// TIA Portal V17 export
// export: Created 2025-03-07T09:19:05.4245713Z, ExportSetting WithDefaults, DisplayName Totally Integrated Automation Portal, DisplayVersion V17 Update 8, DisplayName TIA Portal Openness, DisplayVersion V17 Update 8, DisplayName TIA Portal Version Control Interface, DisplayVersion V17, DisplayName SINAMICS Startdrive Advanced, DisplayVersion V17 SP2, DisplayName SINAMICS Startdrive G110M, G120, G120C, G120D, G120P, G115D, DisplayVersion V17 SP2, DisplayName SINAMICS Startdrive G130, G150, S120, S150, SINAMICS MV, S210, DisplayVersion V17 SP2, DisplayName STEP 7 Professional, DisplayVersion V17 Update 8, DisplayName SINUMERIK ONE STEP 7 Toolbox, DisplayVersion V17 Update 12, DisplayName SINUMERIK 840D sl STEP 7 Toolbox, DisplayVersion V17 Update 12, DisplayName STEP 7 Safety, DisplayVersion V17 Update 6, DisplayName WinCC Advanced, DisplayVersion V17 Update 8
FUNCTION "FC16701_OPC_UA_MASTER_MACHINE_DATA_UPDATE" : Void   // FC16701, LAD
{ S7_Optimized_Access := 'TRUE' }
VERSION : 0.1
// stored: AutoNumber false, IsIECCheckEnabled false, SetENOAutomatically false, UDAEnableTagReadback false
   VAR_TEMP
      RETVAL : Word;
      U01_ASPIRATION_FINAL_VALUE_AUX : Real;
      U02_ASPIRATION_FINAL_VALUE_AUX : Real;
   END_VAR
   VAR_TEMP   // added for the SCL form of the ladder/FBD networks
      _w1 : Bool;
      _w2 : Bool;
      _w3 : Bool;
      _w4 : Bool;
      _w5 : Bool;
   END_VAR
BEGIN

REGION Network 1: <<<<<<<<<<<<<<<<<<<< OPC UA MASTER MACHINE >>>>>>>>>>>>>>>>>>>>
END_REGION

REGION Network 2: GENERAL INFO - ID
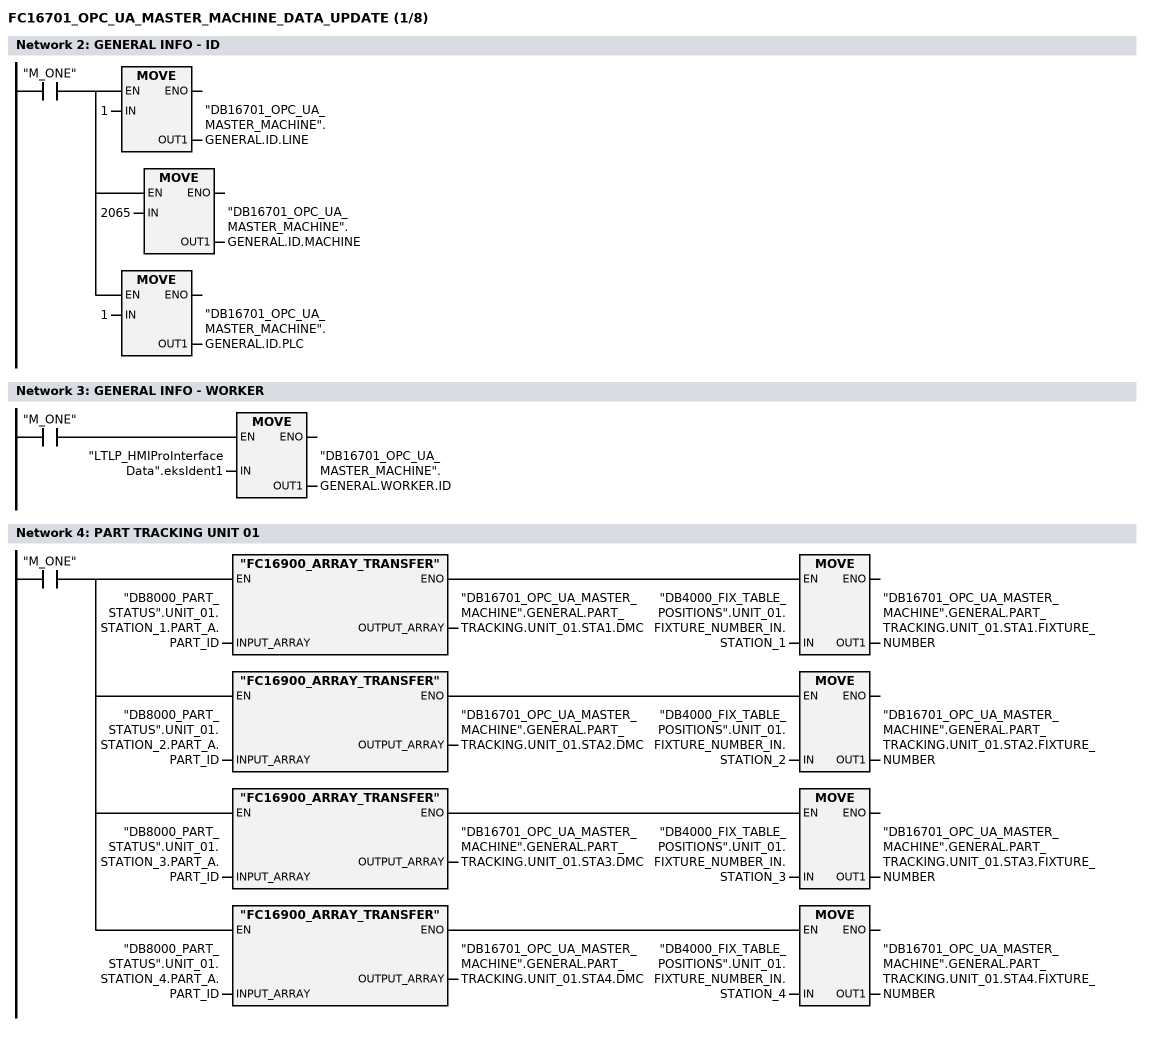
   RUNG wire#powerrail
      Contact( "M_ONE" )
      wire#w1
      Move(in := 1, out1 => "DB16701_OPC_UA_MASTER_MACHINE".GENERAL.ID.LINE)
   END_RUNG
   RUNG wire#w1
      Move(in := 2065, out1 => "DB16701_OPC_UA_MASTER_MACHINE".GENERAL.ID.MACHINE)
   END_RUNG
   RUNG wire#w1
      Move(in := 1, out1 => "DB16701_OPC_UA_MASTER_MACHINE".GENERAL.ID.PLC)
   END_RUNG
   // the same network as SCL:
   IF "M_ONE" THEN
       "DB16701_OPC_UA_MASTER_MACHINE".GENERAL.ID.LINE := 1;
       "DB16701_OPC_UA_MASTER_MACHINE".GENERAL.ID.MACHINE := 2065;
       "DB16701_OPC_UA_MASTER_MACHINE".GENERAL.ID.PLC := 1;
   END_IF;
END_REGION

REGION Network 3: GENERAL INFO - WORKER
   RUNG wire#powerrail
      Contact( "M_ONE" )
      Move(in := "LTLP_HMIProInterfaceData".eksIdent1, out1 => "DB16701_OPC_UA_MASTER_MACHINE".GENERAL.WORKER.ID)
   END_RUNG
   // the same network as SCL:
   IF "M_ONE" THEN
       "DB16701_OPC_UA_MASTER_MACHINE".GENERAL.WORKER.ID := "LTLP_HMIProInterfaceData".eksIdent1;
   END_IF;
END_REGION

REGION Network 4: PART TRACKING UNIT 01
   RUNG wire#powerrail
      Contact( "M_ONE" )
      wire#w1
      "FC16900_ARRAY_TRANSFER"(INPUT_ARRAY := "DB8000_PART_STATUS".UNIT_01.STATION_1.PART_A.PART_ID, OUTPUT_ARRAY => "DB16701_OPC_UA_MASTER_MACHINE".GENERAL.PART_TRACKING.UNIT_01.STA1.DMC)
      Move(in := "DB4000_FIX_TABLE_POSITIONS".UNIT_01.FIXTURE_NUMBER_IN.STATION_1, out1 => "DB16701_OPC_UA_MASTER_MACHINE".GENERAL.PART_TRACKING.UNIT_01.STA1.FIXTURE_NUMBER)
   END_RUNG
   RUNG wire#w1
      "FC16900_ARRAY_TRANSFER"(INPUT_ARRAY := "DB8000_PART_STATUS".UNIT_01.STATION_2.PART_A.PART_ID, OUTPUT_ARRAY => "DB16701_OPC_UA_MASTER_MACHINE".GENERAL.PART_TRACKING.UNIT_01.STA2.DMC)
      Move(in := "DB4000_FIX_TABLE_POSITIONS".UNIT_01.FIXTURE_NUMBER_IN.STATION_2, out1 => "DB16701_OPC_UA_MASTER_MACHINE".GENERAL.PART_TRACKING.UNIT_01.STA2.FIXTURE_NUMBER)
   END_RUNG
   RUNG wire#w1
      "FC16900_ARRAY_TRANSFER"(INPUT_ARRAY := "DB8000_PART_STATUS".UNIT_01.STATION_3.PART_A.PART_ID, OUTPUT_ARRAY => "DB16701_OPC_UA_MASTER_MACHINE".GENERAL.PART_TRACKING.UNIT_01.STA3.DMC)
      Move(in := "DB4000_FIX_TABLE_POSITIONS".UNIT_01.FIXTURE_NUMBER_IN.STATION_3, out1 => "DB16701_OPC_UA_MASTER_MACHINE".GENERAL.PART_TRACKING.UNIT_01.STA3.FIXTURE_NUMBER)
   END_RUNG
   RUNG wire#w1
      "FC16900_ARRAY_TRANSFER"(INPUT_ARRAY := "DB8000_PART_STATUS".UNIT_01.STATION_4.PART_A.PART_ID, OUTPUT_ARRAY => "DB16701_OPC_UA_MASTER_MACHINE".GENERAL.PART_TRACKING.UNIT_01.STA4.DMC)
      Move(in := "DB4000_FIX_TABLE_POSITIONS".UNIT_01.FIXTURE_NUMBER_IN.STATION_4, out1 => "DB16701_OPC_UA_MASTER_MACHINE".GENERAL.PART_TRACKING.UNIT_01.STA4.FIXTURE_NUMBER)
   END_RUNG
   // the same network as SCL:
   #_w2 := "M_ONE";
   "FC16900_ARRAY_TRANSFER"(EN := "M_ONE",
                           INPUT_ARRAY := "DB8000_PART_STATUS".UNIT_01.STATION_1.PART_A.PART_ID,
                           OUTPUT_ARRAY => "DB16701_OPC_UA_MASTER_MACHINE".GENERAL.PART_TRACKING.UNIT_01.STA1.DMC,
                           ENO => #_w1);
   IF #_w1 THEN
       "DB16701_OPC_UA_MASTER_MACHINE".GENERAL.PART_TRACKING.UNIT_01.STA1.FIXTURE_NUMBER := "DB4000_FIX_TABLE_POSITIONS".UNIT_01.FIXTURE_NUMBER_IN.STATION_1;
   END_IF;
   "FC16900_ARRAY_TRANSFER"(EN := #_w2,
                           INPUT_ARRAY := "DB8000_PART_STATUS".UNIT_01.STATION_2.PART_A.PART_ID,
                           OUTPUT_ARRAY => "DB16701_OPC_UA_MASTER_MACHINE".GENERAL.PART_TRACKING.UNIT_01.STA2.DMC,
                           ENO => #_w3);
   IF #_w3 THEN
       "DB16701_OPC_UA_MASTER_MACHINE".GENERAL.PART_TRACKING.UNIT_01.STA2.FIXTURE_NUMBER := "DB4000_FIX_TABLE_POSITIONS".UNIT_01.FIXTURE_NUMBER_IN.STATION_2;
   END_IF;
   "FC16900_ARRAY_TRANSFER"(EN := #_w2,
                           INPUT_ARRAY := "DB8000_PART_STATUS".UNIT_01.STATION_3.PART_A.PART_ID,
                           OUTPUT_ARRAY => "DB16701_OPC_UA_MASTER_MACHINE".GENERAL.PART_TRACKING.UNIT_01.STA3.DMC,
                           ENO => #_w4);
   IF #_w4 THEN
       "DB16701_OPC_UA_MASTER_MACHINE".GENERAL.PART_TRACKING.UNIT_01.STA3.FIXTURE_NUMBER := "DB4000_FIX_TABLE_POSITIONS".UNIT_01.FIXTURE_NUMBER_IN.STATION_3;
   END_IF;
   "FC16900_ARRAY_TRANSFER"(EN := #_w2,
                           INPUT_ARRAY := "DB8000_PART_STATUS".UNIT_01.STATION_4.PART_A.PART_ID,
                           OUTPUT_ARRAY => "DB16701_OPC_UA_MASTER_MACHINE".GENERAL.PART_TRACKING.UNIT_01.STA4.DMC,
                           ENO => #_w5);
   IF #_w5 THEN
       "DB16701_OPC_UA_MASTER_MACHINE".GENERAL.PART_TRACKING.UNIT_01.STA4.FIXTURE_NUMBER := "DB4000_FIX_TABLE_POSITIONS".UNIT_01.FIXTURE_NUMBER_IN.STATION_4;
   END_IF;
END_REGION

REGION Network 5: PART TRACKING UNIT 02
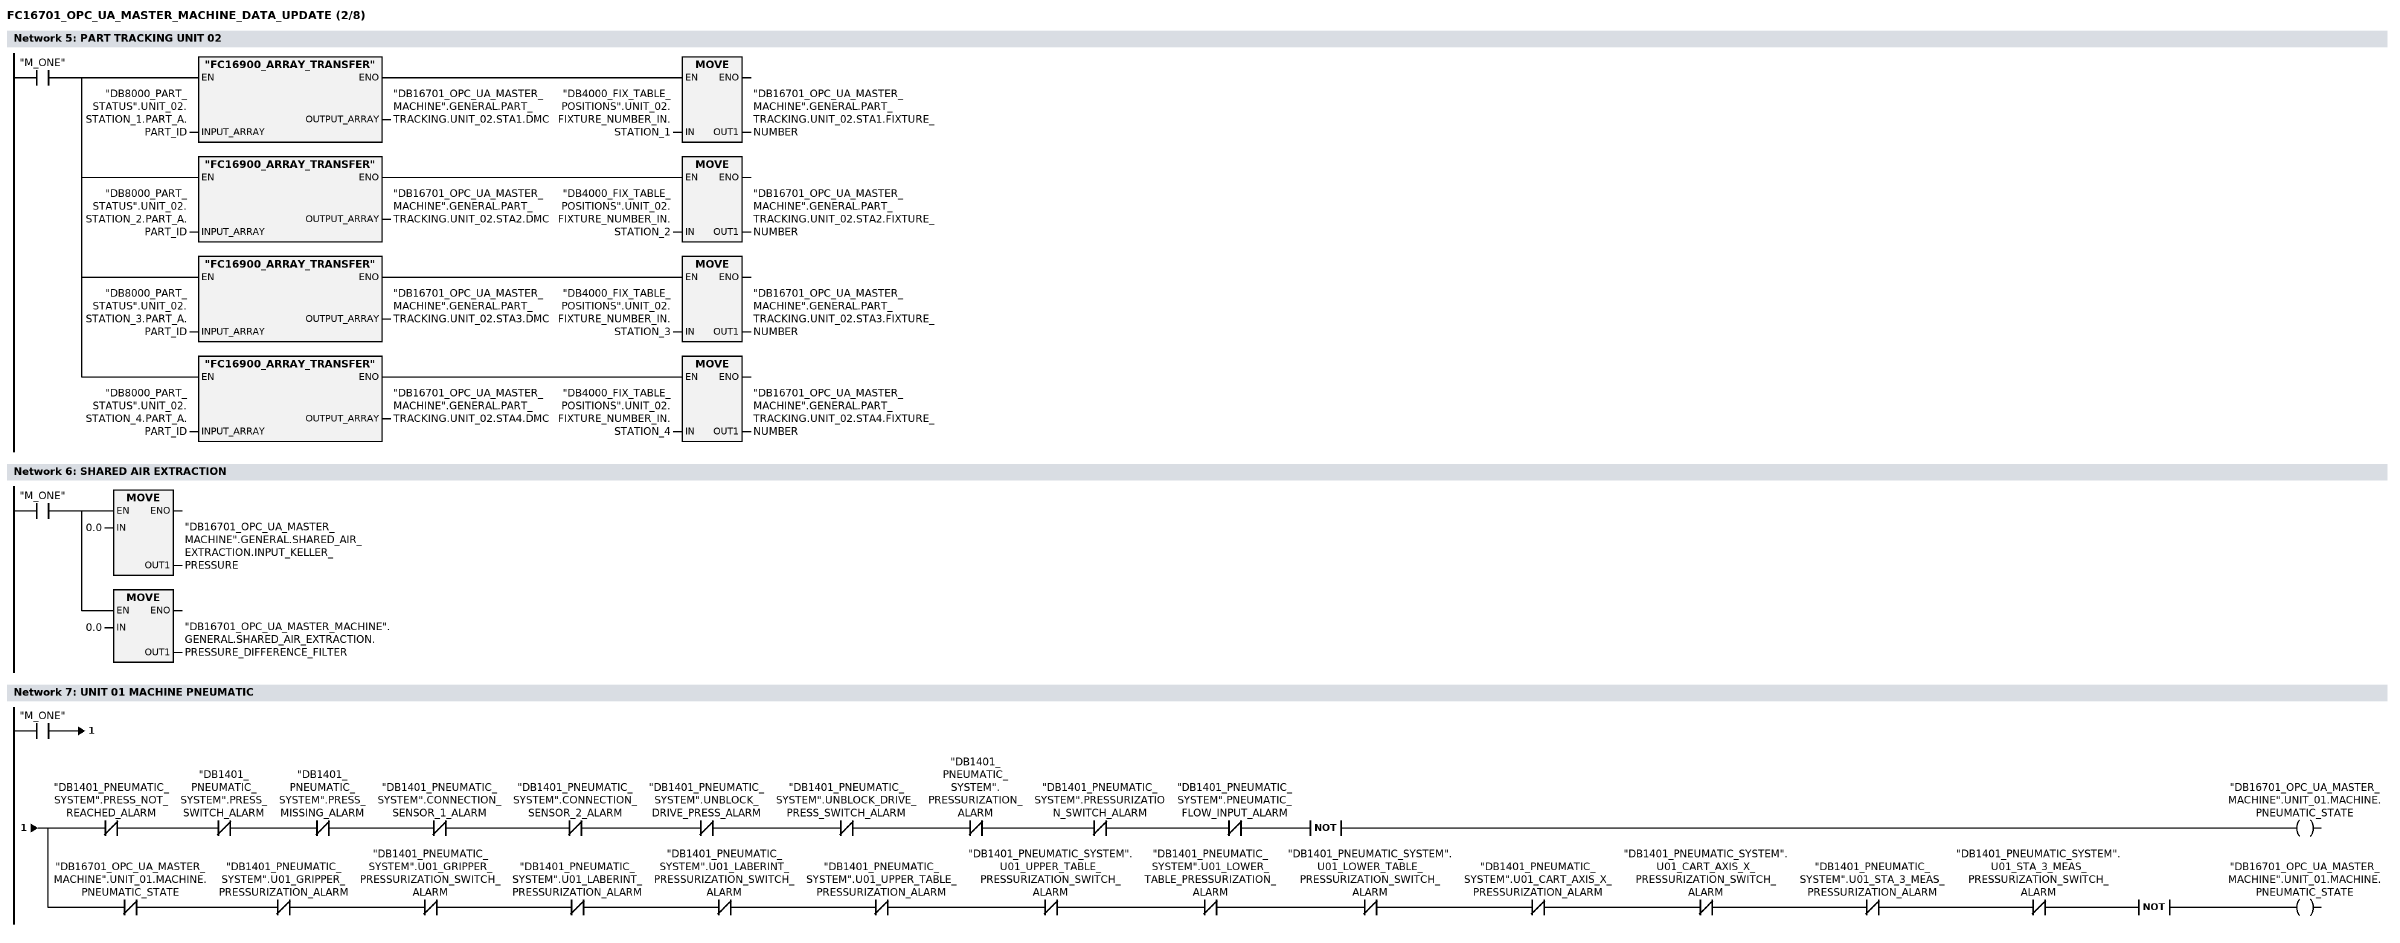
   RUNG wire#powerrail
      Contact( "M_ONE" )
      wire#w1
      "FC16900_ARRAY_TRANSFER"(INPUT_ARRAY := "DB8000_PART_STATUS".UNIT_02.STATION_1.PART_A.PART_ID, OUTPUT_ARRAY => "DB16701_OPC_UA_MASTER_MACHINE".GENERAL.PART_TRACKING.UNIT_02.STA1.DMC)
      Move(in := "DB4000_FIX_TABLE_POSITIONS".UNIT_02.FIXTURE_NUMBER_IN.STATION_1, out1 => "DB16701_OPC_UA_MASTER_MACHINE".GENERAL.PART_TRACKING.UNIT_02.STA1.FIXTURE_NUMBER)
   END_RUNG
   RUNG wire#w1
      "FC16900_ARRAY_TRANSFER"(INPUT_ARRAY := "DB8000_PART_STATUS".UNIT_02.STATION_2.PART_A.PART_ID, OUTPUT_ARRAY => "DB16701_OPC_UA_MASTER_MACHINE".GENERAL.PART_TRACKING.UNIT_02.STA2.DMC)
      Move(in := "DB4000_FIX_TABLE_POSITIONS".UNIT_02.FIXTURE_NUMBER_IN.STATION_2, out1 => "DB16701_OPC_UA_MASTER_MACHINE".GENERAL.PART_TRACKING.UNIT_02.STA2.FIXTURE_NUMBER)
   END_RUNG
   RUNG wire#w1
      "FC16900_ARRAY_TRANSFER"(INPUT_ARRAY := "DB8000_PART_STATUS".UNIT_02.STATION_3.PART_A.PART_ID, OUTPUT_ARRAY => "DB16701_OPC_UA_MASTER_MACHINE".GENERAL.PART_TRACKING.UNIT_02.STA3.DMC)
      Move(in := "DB4000_FIX_TABLE_POSITIONS".UNIT_02.FIXTURE_NUMBER_IN.STATION_3, out1 => "DB16701_OPC_UA_MASTER_MACHINE".GENERAL.PART_TRACKING.UNIT_02.STA3.FIXTURE_NUMBER)
   END_RUNG
   RUNG wire#w1
      "FC16900_ARRAY_TRANSFER"(INPUT_ARRAY := "DB8000_PART_STATUS".UNIT_02.STATION_4.PART_A.PART_ID, OUTPUT_ARRAY => "DB16701_OPC_UA_MASTER_MACHINE".GENERAL.PART_TRACKING.UNIT_02.STA4.DMC)
      Move(in := "DB4000_FIX_TABLE_POSITIONS".UNIT_02.FIXTURE_NUMBER_IN.STATION_4, out1 => "DB16701_OPC_UA_MASTER_MACHINE".GENERAL.PART_TRACKING.UNIT_02.STA4.FIXTURE_NUMBER)
   END_RUNG
   // the same network as SCL:
   #_w2 := "M_ONE";
   "FC16900_ARRAY_TRANSFER"(EN := "M_ONE",
                           INPUT_ARRAY := "DB8000_PART_STATUS".UNIT_02.STATION_1.PART_A.PART_ID,
                           OUTPUT_ARRAY => "DB16701_OPC_UA_MASTER_MACHINE".GENERAL.PART_TRACKING.UNIT_02.STA1.DMC,
                           ENO => #_w1);
   IF #_w1 THEN
       "DB16701_OPC_UA_MASTER_MACHINE".GENERAL.PART_TRACKING.UNIT_02.STA1.FIXTURE_NUMBER := "DB4000_FIX_TABLE_POSITIONS".UNIT_02.FIXTURE_NUMBER_IN.STATION_1;
   END_IF;
   "FC16900_ARRAY_TRANSFER"(EN := #_w2,
                           INPUT_ARRAY := "DB8000_PART_STATUS".UNIT_02.STATION_2.PART_A.PART_ID,
                           OUTPUT_ARRAY => "DB16701_OPC_UA_MASTER_MACHINE".GENERAL.PART_TRACKING.UNIT_02.STA2.DMC,
                           ENO => #_w3);
   IF #_w3 THEN
       "DB16701_OPC_UA_MASTER_MACHINE".GENERAL.PART_TRACKING.UNIT_02.STA2.FIXTURE_NUMBER := "DB4000_FIX_TABLE_POSITIONS".UNIT_02.FIXTURE_NUMBER_IN.STATION_2;
   END_IF;
   "FC16900_ARRAY_TRANSFER"(EN := #_w2,
                           INPUT_ARRAY := "DB8000_PART_STATUS".UNIT_02.STATION_3.PART_A.PART_ID,
                           OUTPUT_ARRAY => "DB16701_OPC_UA_MASTER_MACHINE".GENERAL.PART_TRACKING.UNIT_02.STA3.DMC,
                           ENO => #_w4);
   IF #_w4 THEN
       "DB16701_OPC_UA_MASTER_MACHINE".GENERAL.PART_TRACKING.UNIT_02.STA3.FIXTURE_NUMBER := "DB4000_FIX_TABLE_POSITIONS".UNIT_02.FIXTURE_NUMBER_IN.STATION_3;
   END_IF;
   "FC16900_ARRAY_TRANSFER"(EN := #_w2,
                           INPUT_ARRAY := "DB8000_PART_STATUS".UNIT_02.STATION_4.PART_A.PART_ID,
                           OUTPUT_ARRAY => "DB16701_OPC_UA_MASTER_MACHINE".GENERAL.PART_TRACKING.UNIT_02.STA4.DMC,
                           ENO => #_w5);
   IF #_w5 THEN
       "DB16701_OPC_UA_MASTER_MACHINE".GENERAL.PART_TRACKING.UNIT_02.STA4.FIXTURE_NUMBER := "DB4000_FIX_TABLE_POSITIONS".UNIT_02.FIXTURE_NUMBER_IN.STATION_4;
   END_IF;
END_REGION

REGION Network 6: SHARED AIR EXTRACTION
   RUNG wire#powerrail
      Contact( "M_ONE" )
      wire#w1
      Move(in := 0.0, out1 => "DB16701_OPC_UA_MASTER_MACHINE".GENERAL.SHARED_AIR_EXTRACTION.INPUT_KELLER_PRESSURE)
   END_RUNG
   RUNG wire#w1
      Move(in := 0.0, out1 => "DB16701_OPC_UA_MASTER_MACHINE".GENERAL.SHARED_AIR_EXTRACTION.PRESSURE_DIFFERENCE_FILTER)
   END_RUNG
   // the same network as SCL:
   IF "M_ONE" THEN
       "DB16701_OPC_UA_MASTER_MACHINE".GENERAL.SHARED_AIR_EXTRACTION.INPUT_KELLER_PRESSURE := 0.0;
       "DB16701_OPC_UA_MASTER_MACHINE".GENERAL.SHARED_AIR_EXTRACTION.PRESSURE_DIFFERENCE_FILTER := 0.0;
   END_IF;
END_REGION

REGION Network 7: UNIT 01 MACHINE PNEUMATIC
   RUNG wire#powerrail
      Contact( "M_ONE" )
      wire#w1
      I_Contact( "DB1401_PNEUMATIC_SYSTEM".PRESS_NOT_REACHED_ALARM )
      I_Contact( "DB1401_PNEUMATIC_SYSTEM".PRESS_SWITCH_ALARM )
      I_Contact( "DB1401_PNEUMATIC_SYSTEM".PRESS_MISSING_ALARM )
      I_Contact( "DB1401_PNEUMATIC_SYSTEM".CONNECTION_SENSOR_1_ALARM )
      I_Contact( "DB1401_PNEUMATIC_SYSTEM".CONNECTION_SENSOR_2_ALARM )
      I_Contact( "DB1401_PNEUMATIC_SYSTEM".UNBLOCK_DRIVE_PRESS_ALARM )
      I_Contact( "DB1401_PNEUMATIC_SYSTEM".UNBLOCK_DRIVE_PRESS_SWITCH_ALARM )
      I_Contact( "DB1401_PNEUMATIC_SYSTEM".PRESSURIZATION_ALARM )
      I_Contact( "DB1401_PNEUMATIC_SYSTEM".PRESSURIZATION_SWITCH_ALARM )
      I_Contact( "DB1401_PNEUMATIC_SYSTEM".PNEUMATIC_FLOW_INPUT_ALARM )
      Not()
      Coil( "DB16701_OPC_UA_MASTER_MACHINE".UNIT_01.MACHINE.PNEUMATIC_STATE )
   END_RUNG
   RUNG wire#w1
      I_Contact( "DB16701_OPC_UA_MASTER_MACHINE".UNIT_01.MACHINE.PNEUMATIC_STATE )
      I_Contact( "DB1401_PNEUMATIC_SYSTEM".U01_GRIPPER_PRESSURIZATION_ALARM )
      I_Contact( "DB1401_PNEUMATIC_SYSTEM".U01_GRIPPER_PRESSURIZATION_SWITCH_ALARM )
      I_Contact( "DB1401_PNEUMATIC_SYSTEM".U01_LABERINT_PRESSURIZATION_ALARM )
      I_Contact( "DB1401_PNEUMATIC_SYSTEM".U01_LABERINT_PRESSURIZATION_SWITCH_ALARM )
      I_Contact( "DB1401_PNEUMATIC_SYSTEM".U01_UPPER_TABLE_PRESSURIZATION_ALARM )
      I_Contact( "DB1401_PNEUMATIC_SYSTEM".U01_UPPER_TABLE_PRESSURIZATION_SWITCH_ALARM )
      I_Contact( "DB1401_PNEUMATIC_SYSTEM".U01_LOWER_TABLE_PRESSURIZATION_ALARM )
      I_Contact( "DB1401_PNEUMATIC_SYSTEM".U01_LOWER_TABLE_PRESSURIZATION_SWITCH_ALARM )
      I_Contact( "DB1401_PNEUMATIC_SYSTEM".U01_CART_AXIS_X_PRESSURIZATION_ALARM )
      I_Contact( "DB1401_PNEUMATIC_SYSTEM".U01_CART_AXIS_X_PRESSURIZATION_SWITCH_ALARM )
      I_Contact( "DB1401_PNEUMATIC_SYSTEM".U01_STA_3_MEAS_PRESSURIZATION_ALARM )
      I_Contact( "DB1401_PNEUMATIC_SYSTEM".U01_STA_3_MEAS_PRESSURIZATION_SWITCH_ALARM )
      Not()
      Coil( "DB16701_OPC_UA_MASTER_MACHINE".UNIT_01.MACHINE.PNEUMATIC_STATE )
   END_RUNG
   // the same network as SCL:
   "DB16701_OPC_UA_MASTER_MACHINE".UNIT_01.MACHINE.PNEUMATIC_STATE := NOT ("M_ONE" AND NOT "DB1401_PNEUMATIC_SYSTEM".PRESS_NOT_REACHED_ALARM AND NOT "DB1401_PNEUMATIC_SYSTEM".PRESS_SWITCH_ALARM AND NOT "DB1401_PNEUMATIC_SYSTEM".PRESS_MISSING_ALARM AND NOT "DB1401_PNEUMATIC_SYSTEM".CONNECTION_SENSOR_1_ALARM AND NOT "DB1401_PNEUMATIC_SYSTEM".CONNECTION_SENSOR_2_ALARM AND NOT "DB1401_PNEUMATIC_SYSTEM".UNBLOCK_DRIVE_PRESS_ALARM AND NOT "DB1401_PNEUMATIC_SYSTEM".UNBLOCK_DRIVE_PRESS_SWITCH_ALARM AND NOT "DB1401_PNEUMATIC_SYSTEM".PRESSURIZATION_ALARM AND NOT "DB1401_PNEUMATIC_SYSTEM".PRESSURIZATION_SWITCH_ALARM AND NOT "DB1401_PNEUMATIC_SYSTEM".PNEUMATIC_FLOW_INPUT_ALARM);
   "DB16701_OPC_UA_MASTER_MACHINE".UNIT_01.MACHINE.PNEUMATIC_STATE := NOT ("M_ONE" AND NOT "DB16701_OPC_UA_MASTER_MACHINE".UNIT_01.MACHINE.PNEUMATIC_STATE AND NOT "DB1401_PNEUMATIC_SYSTEM".U01_GRIPPER_PRESSURIZATION_ALARM AND NOT "DB1401_PNEUMATIC_SYSTEM".U01_GRIPPER_PRESSURIZATION_SWITCH_ALARM AND NOT "DB1401_PNEUMATIC_SYSTEM".U01_LABERINT_PRESSURIZATION_ALARM AND NOT "DB1401_PNEUMATIC_SYSTEM".U01_LABERINT_PRESSURIZATION_SWITCH_ALARM AND NOT "DB1401_PNEUMATIC_SYSTEM".U01_UPPER_TABLE_PRESSURIZATION_ALARM AND NOT "DB1401_PNEUMATIC_SYSTEM".U01_UPPER_TABLE_PRESSURIZATION_SWITCH_ALARM AND NOT "DB1401_PNEUMATIC_SYSTEM".U01_LOWER_TABLE_PRESSURIZATION_ALARM AND NOT "DB1401_PNEUMATIC_SYSTEM".U01_LOWER_TABLE_PRESSURIZATION_SWITCH_ALARM AND NOT "DB1401_PNEUMATIC_SYSTEM".U01_CART_AXIS_X_PRESSURIZATION_ALARM AND NOT "DB1401_PNEUMATIC_SYSTEM".U01_CART_AXIS_X_PRESSURIZATION_SWITCH_ALARM AND NOT "DB1401_PNEUMATIC_SYSTEM".U01_STA_3_MEAS_PRESSURIZATION_ALARM AND NOT "DB1401_PNEUMATIC_SYSTEM".U01_STA_3_MEAS_PRESSURIZATION_SWITCH_ALARM);
END_REGION

REGION Network 8: UNIT 01 MACHINE TEMPERATURE
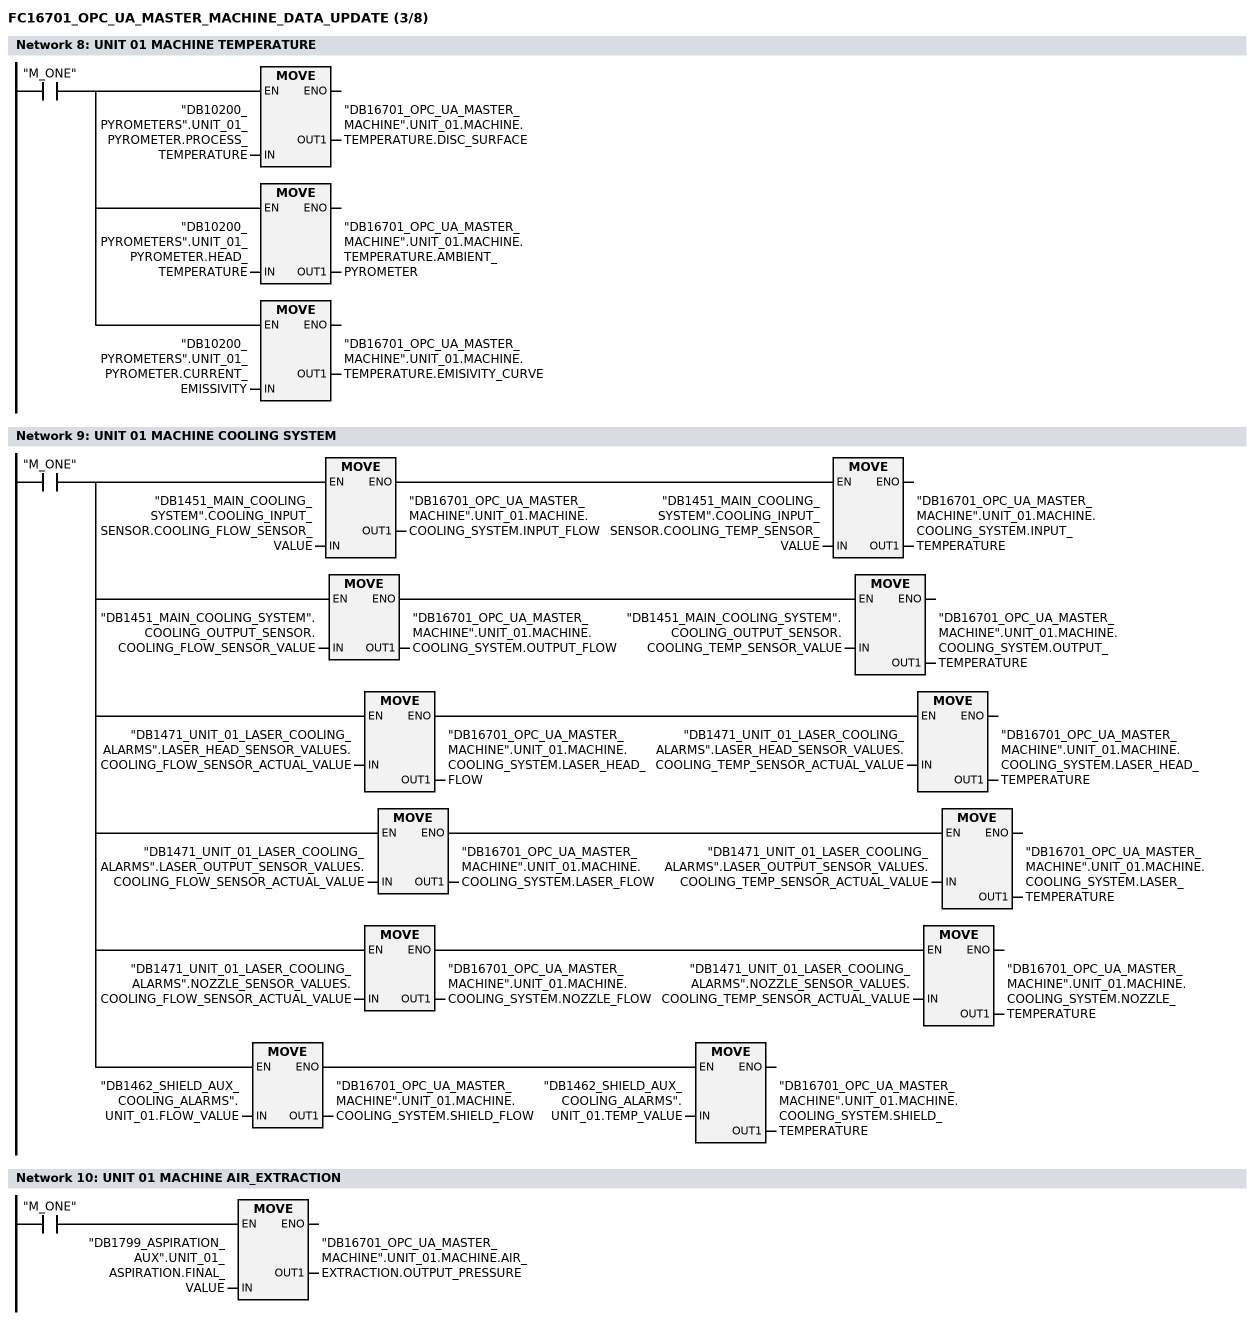
   RUNG wire#powerrail
      Contact( "M_ONE" )
      wire#w1
      Move(in := "DB10200_PYROMETERS".UNIT_01_PYROMETER.PROCESS_TEMPERATURE, out1 => "DB16701_OPC_UA_MASTER_MACHINE".UNIT_01.MACHINE.TEMPERATURE.DISC_SURFACE)
   END_RUNG
   RUNG wire#w1
      Move(in := "DB10200_PYROMETERS".UNIT_01_PYROMETER.HEAD_TEMPERATURE, out1 => "DB16701_OPC_UA_MASTER_MACHINE".UNIT_01.MACHINE.TEMPERATURE.AMBIENT_PYROMETER)
   END_RUNG
   RUNG wire#w1
      Move(in := "DB10200_PYROMETERS".UNIT_01_PYROMETER.CURRENT_EMISSIVITY, out1 => "DB16701_OPC_UA_MASTER_MACHINE".UNIT_01.MACHINE.TEMPERATURE.EMISIVITY_CURVE)
   END_RUNG
   // the same network as SCL:
   IF "M_ONE" THEN
       "DB16701_OPC_UA_MASTER_MACHINE".UNIT_01.MACHINE.TEMPERATURE.DISC_SURFACE := "DB10200_PYROMETERS".UNIT_01_PYROMETER.PROCESS_TEMPERATURE;
       "DB16701_OPC_UA_MASTER_MACHINE".UNIT_01.MACHINE.TEMPERATURE.AMBIENT_PYROMETER := "DB10200_PYROMETERS".UNIT_01_PYROMETER.HEAD_TEMPERATURE;
       "DB16701_OPC_UA_MASTER_MACHINE".UNIT_01.MACHINE.TEMPERATURE.EMISIVITY_CURVE := "DB10200_PYROMETERS".UNIT_01_PYROMETER.CURRENT_EMISSIVITY;
   END_IF;
END_REGION

REGION Network 9: UNIT 01 MACHINE COOLING SYSTEM
   RUNG wire#powerrail
      Contact( "M_ONE" )
      wire#w1
      Move(in := "DB1451_MAIN_COOLING_SYSTEM".COOLING_INPUT_SENSOR.COOLING_FLOW_SENSOR_VALUE, out1 => "DB16701_OPC_UA_MASTER_MACHINE".UNIT_01.MACHINE.COOLING_SYSTEM.INPUT_FLOW)
      Move(in := "DB1451_MAIN_COOLING_SYSTEM".COOLING_INPUT_SENSOR.COOLING_TEMP_SENSOR_VALUE, out1 => "DB16701_OPC_UA_MASTER_MACHINE".UNIT_01.MACHINE.COOLING_SYSTEM.INPUT_TEMPERATURE)
   END_RUNG
   RUNG wire#w1
      Move(in := "DB1451_MAIN_COOLING_SYSTEM".COOLING_OUTPUT_SENSOR.COOLING_FLOW_SENSOR_VALUE, out1 => "DB16701_OPC_UA_MASTER_MACHINE".UNIT_01.MACHINE.COOLING_SYSTEM.OUTPUT_FLOW)
      Move(in := "DB1451_MAIN_COOLING_SYSTEM".COOLING_OUTPUT_SENSOR.COOLING_TEMP_SENSOR_VALUE, out1 => "DB16701_OPC_UA_MASTER_MACHINE".UNIT_01.MACHINE.COOLING_SYSTEM.OUTPUT_TEMPERATURE)
   END_RUNG
   RUNG wire#w1
      Move(in := "DB1471_UNIT_01_LASER_COOLING_ALARMS".LASER_HEAD_SENSOR_VALUES.COOLING_FLOW_SENSOR_ACTUAL_VALUE, out1 => "DB16701_OPC_UA_MASTER_MACHINE".UNIT_01.MACHINE.COOLING_SYSTEM.LASER_HEAD_FLOW)
      Move(in := "DB1471_UNIT_01_LASER_COOLING_ALARMS".LASER_HEAD_SENSOR_VALUES.COOLING_TEMP_SENSOR_ACTUAL_VALUE, out1 => "DB16701_OPC_UA_MASTER_MACHINE".UNIT_01.MACHINE.COOLING_SYSTEM.LASER_HEAD_TEMPERATURE)
   END_RUNG
   RUNG wire#w1
      Move(in := "DB1471_UNIT_01_LASER_COOLING_ALARMS".LASER_OUTPUT_SENSOR_VALUES.COOLING_FLOW_SENSOR_ACTUAL_VALUE, out1 => "DB16701_OPC_UA_MASTER_MACHINE".UNIT_01.MACHINE.COOLING_SYSTEM.LASER_FLOW)
      Move(in := "DB1471_UNIT_01_LASER_COOLING_ALARMS".LASER_OUTPUT_SENSOR_VALUES.COOLING_TEMP_SENSOR_ACTUAL_VALUE, out1 => "DB16701_OPC_UA_MASTER_MACHINE".UNIT_01.MACHINE.COOLING_SYSTEM.LASER_TEMPERATURE)
   END_RUNG
   RUNG wire#w1
      Move(in := "DB1471_UNIT_01_LASER_COOLING_ALARMS".NOZZLE_SENSOR_VALUES.COOLING_FLOW_SENSOR_ACTUAL_VALUE, out1 => "DB16701_OPC_UA_MASTER_MACHINE".UNIT_01.MACHINE.COOLING_SYSTEM.NOZZLE_FLOW)
      Move(in := "DB1471_UNIT_01_LASER_COOLING_ALARMS".NOZZLE_SENSOR_VALUES.COOLING_TEMP_SENSOR_ACTUAL_VALUE, out1 => "DB16701_OPC_UA_MASTER_MACHINE".UNIT_01.MACHINE.COOLING_SYSTEM.NOZZLE_TEMPERATURE)
   END_RUNG
   RUNG wire#w1
      Move(in := "DB1462_SHIELD_AUX_COOLING_ALARMS".UNIT_01.FLOW_VALUE, out1 => "DB16701_OPC_UA_MASTER_MACHINE".UNIT_01.MACHINE.COOLING_SYSTEM.SHIELD_FLOW)
      Move(in := "DB1462_SHIELD_AUX_COOLING_ALARMS".UNIT_01.TEMP_VALUE, out1 => "DB16701_OPC_UA_MASTER_MACHINE".UNIT_01.MACHINE.COOLING_SYSTEM.SHIELD_TEMPERATURE)
   END_RUNG
   // the same network as SCL:
   IF "M_ONE" THEN
       "DB16701_OPC_UA_MASTER_MACHINE".UNIT_01.MACHINE.COOLING_SYSTEM.INPUT_FLOW := "DB1451_MAIN_COOLING_SYSTEM".COOLING_INPUT_SENSOR.COOLING_FLOW_SENSOR_VALUE;
       "DB16701_OPC_UA_MASTER_MACHINE".UNIT_01.MACHINE.COOLING_SYSTEM.INPUT_TEMPERATURE := "DB1451_MAIN_COOLING_SYSTEM".COOLING_INPUT_SENSOR.COOLING_TEMP_SENSOR_VALUE;
       "DB16701_OPC_UA_MASTER_MACHINE".UNIT_01.MACHINE.COOLING_SYSTEM.OUTPUT_FLOW := "DB1451_MAIN_COOLING_SYSTEM".COOLING_OUTPUT_SENSOR.COOLING_FLOW_SENSOR_VALUE;
       "DB16701_OPC_UA_MASTER_MACHINE".UNIT_01.MACHINE.COOLING_SYSTEM.OUTPUT_TEMPERATURE := "DB1451_MAIN_COOLING_SYSTEM".COOLING_OUTPUT_SENSOR.COOLING_TEMP_SENSOR_VALUE;
       "DB16701_OPC_UA_MASTER_MACHINE".UNIT_01.MACHINE.COOLING_SYSTEM.LASER_HEAD_FLOW := "DB1471_UNIT_01_LASER_COOLING_ALARMS".LASER_HEAD_SENSOR_VALUES.COOLING_FLOW_SENSOR_ACTUAL_VALUE;
       "DB16701_OPC_UA_MASTER_MACHINE".UNIT_01.MACHINE.COOLING_SYSTEM.LASER_HEAD_TEMPERATURE := "DB1471_UNIT_01_LASER_COOLING_ALARMS".LASER_HEAD_SENSOR_VALUES.COOLING_TEMP_SENSOR_ACTUAL_VALUE;
       "DB16701_OPC_UA_MASTER_MACHINE".UNIT_01.MACHINE.COOLING_SYSTEM.LASER_FLOW := "DB1471_UNIT_01_LASER_COOLING_ALARMS".LASER_OUTPUT_SENSOR_VALUES.COOLING_FLOW_SENSOR_ACTUAL_VALUE;
       "DB16701_OPC_UA_MASTER_MACHINE".UNIT_01.MACHINE.COOLING_SYSTEM.LASER_TEMPERATURE := "DB1471_UNIT_01_LASER_COOLING_ALARMS".LASER_OUTPUT_SENSOR_VALUES.COOLING_TEMP_SENSOR_ACTUAL_VALUE;
       "DB16701_OPC_UA_MASTER_MACHINE".UNIT_01.MACHINE.COOLING_SYSTEM.NOZZLE_FLOW := "DB1471_UNIT_01_LASER_COOLING_ALARMS".NOZZLE_SENSOR_VALUES.COOLING_FLOW_SENSOR_ACTUAL_VALUE;
       "DB16701_OPC_UA_MASTER_MACHINE".UNIT_01.MACHINE.COOLING_SYSTEM.NOZZLE_TEMPERATURE := "DB1471_UNIT_01_LASER_COOLING_ALARMS".NOZZLE_SENSOR_VALUES.COOLING_TEMP_SENSOR_ACTUAL_VALUE;
       "DB16701_OPC_UA_MASTER_MACHINE".UNIT_01.MACHINE.COOLING_SYSTEM.SHIELD_FLOW := "DB1462_SHIELD_AUX_COOLING_ALARMS".UNIT_01.FLOW_VALUE;
       "DB16701_OPC_UA_MASTER_MACHINE".UNIT_01.MACHINE.COOLING_SYSTEM.SHIELD_TEMPERATURE := "DB1462_SHIELD_AUX_COOLING_ALARMS".UNIT_01.TEMP_VALUE;
   END_IF;
END_REGION

REGION Network 10: UNIT 01 MACHINE AIR_EXTRACTION
   RUNG wire#powerrail
      Contact( "M_ONE" )
      Move(in := "DB1799_ASPIRATION_AUX".UNIT_01_ASPIRATION.FINAL_VALUE, out1 => "DB16701_OPC_UA_MASTER_MACHINE".UNIT_01.MACHINE.AIR_EXTRACTION.OUTPUT_PRESSURE)
   END_RUNG
   // the same network as SCL:
   IF "M_ONE" THEN
       "DB16701_OPC_UA_MASTER_MACHINE".UNIT_01.MACHINE.AIR_EXTRACTION.OUTPUT_PRESSURE := "DB1799_ASPIRATION_AUX".UNIT_01_ASPIRATION.FINAL_VALUE;
   END_IF;
END_REGION

REGION Network 11: UNIT 01 MACHINE ST3 PRESSURE CONTROL
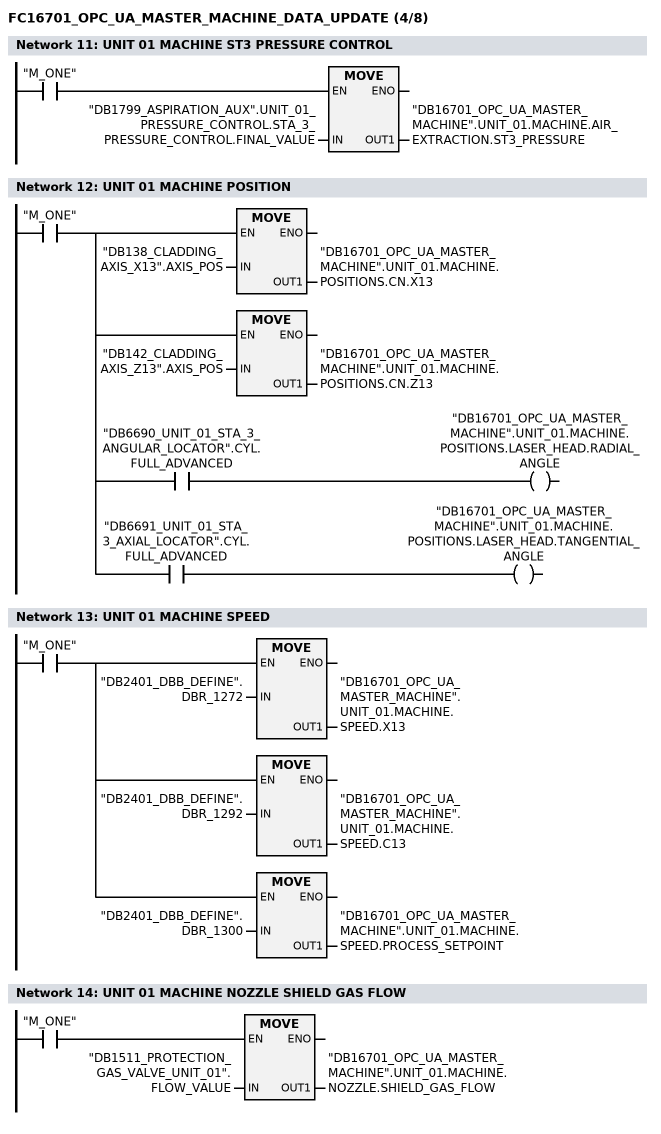
   RUNG wire#powerrail
      Contact( "M_ONE" )
      Move(in := "DB1799_ASPIRATION_AUX".UNIT_01_PRESSURE_CONTROL.STA_3_PRESSURE_CONTROL.FINAL_VALUE, out1 => "DB16701_OPC_UA_MASTER_MACHINE".UNIT_01.MACHINE.AIR_EXTRACTION.ST3_PRESSURE)
   END_RUNG
   // the same network as SCL:
   IF "M_ONE" THEN
       "DB16701_OPC_UA_MASTER_MACHINE".UNIT_01.MACHINE.AIR_EXTRACTION.ST3_PRESSURE := "DB1799_ASPIRATION_AUX".UNIT_01_PRESSURE_CONTROL.STA_3_PRESSURE_CONTROL.FINAL_VALUE;
   END_IF;
END_REGION

REGION Network 12: UNIT 01 MACHINE POSITION
   RUNG wire#powerrail
      Contact( "M_ONE" )
      wire#w1
      Move(in := "DB138_CLADDING_AXIS_X13".AXIS_POS, out1 => "DB16701_OPC_UA_MASTER_MACHINE".UNIT_01.MACHINE.POSITIONS.CN.X13)
   END_RUNG
   RUNG wire#w1
      Move(in := "DB142_CLADDING_AXIS_Z13".AXIS_POS, out1 => "DB16701_OPC_UA_MASTER_MACHINE".UNIT_01.MACHINE.POSITIONS.CN.Z13)
   END_RUNG
   RUNG wire#w1
      Contact( "DB6690_UNIT_01_STA_3_ANGULAR_LOCATOR".CYL.FULL_ADVANCED )
      Coil( "DB16701_OPC_UA_MASTER_MACHINE".UNIT_01.MACHINE.POSITIONS.LASER_HEAD.RADIAL_ANGLE )
   END_RUNG
   RUNG wire#w1
      Contact( "DB6691_UNIT_01_STA_3_AXIAL_LOCATOR".CYL.FULL_ADVANCED )
      Coil( "DB16701_OPC_UA_MASTER_MACHINE".UNIT_01.MACHINE.POSITIONS.LASER_HEAD.TANGENTIAL_ANGLE )
   END_RUNG
   // the same network as SCL:
   IF "M_ONE" THEN
       "DB16701_OPC_UA_MASTER_MACHINE".UNIT_01.MACHINE.POSITIONS.CN.X13 := "DB138_CLADDING_AXIS_X13".AXIS_POS;
       "DB16701_OPC_UA_MASTER_MACHINE".UNIT_01.MACHINE.POSITIONS.CN.Z13 := "DB142_CLADDING_AXIS_Z13".AXIS_POS;
   END_IF;
   "DB16701_OPC_UA_MASTER_MACHINE".UNIT_01.MACHINE.POSITIONS.LASER_HEAD.RADIAL_ANGLE := "M_ONE" AND "DB6690_UNIT_01_STA_3_ANGULAR_LOCATOR".CYL.FULL_ADVANCED;
   "DB16701_OPC_UA_MASTER_MACHINE".UNIT_01.MACHINE.POSITIONS.LASER_HEAD.TANGENTIAL_ANGLE := "M_ONE" AND "DB6691_UNIT_01_STA_3_AXIAL_LOCATOR".CYL.FULL_ADVANCED;
END_REGION

REGION Network 13: UNIT 01 MACHINE SPEED
   RUNG wire#powerrail
      Contact( "M_ONE" )
      wire#w1
      Move(in := "DB2401_DBB_DEFINE".DBR_1272, out1 => "DB16701_OPC_UA_MASTER_MACHINE".UNIT_01.MACHINE.SPEED.X13)
   END_RUNG
   RUNG wire#w1
      Move(in := "DB2401_DBB_DEFINE".DBR_1292, out1 => "DB16701_OPC_UA_MASTER_MACHINE".UNIT_01.MACHINE.SPEED.C13)
   END_RUNG
   RUNG wire#w1
      Move(in := "DB2401_DBB_DEFINE".DBR_1300, out1 => "DB16701_OPC_UA_MASTER_MACHINE".UNIT_01.MACHINE.SPEED.PROCESS_SETPOINT)
   END_RUNG
   // the same network as SCL:
   IF "M_ONE" THEN
       "DB16701_OPC_UA_MASTER_MACHINE".UNIT_01.MACHINE.SPEED.X13 := "DB2401_DBB_DEFINE".DBR_1272;
       "DB16701_OPC_UA_MASTER_MACHINE".UNIT_01.MACHINE.SPEED.C13 := "DB2401_DBB_DEFINE".DBR_1292;
       "DB16701_OPC_UA_MASTER_MACHINE".UNIT_01.MACHINE.SPEED.PROCESS_SETPOINT := "DB2401_DBB_DEFINE".DBR_1300;
   END_IF;
END_REGION

REGION Network 14: UNIT 01 MACHINE NOZZLE SHIELD GAS FLOW
   RUNG wire#powerrail
      Contact( "M_ONE" )
      Move(in := "DB1511_PROTECTION_GAS_VALVE_UNIT_01".FLOW_VALUE, out1 => "DB16701_OPC_UA_MASTER_MACHINE".UNIT_01.MACHINE.NOZZLE.SHIELD_GAS_FLOW)
   END_RUNG
   // the same network as SCL:
   IF "M_ONE" THEN
       "DB16701_OPC_UA_MASTER_MACHINE".UNIT_01.MACHINE.NOZZLE.SHIELD_GAS_FLOW := "DB1511_PROTECTION_GAS_VALVE_UNIT_01".FLOW_VALUE;
   END_IF;
END_REGION

REGION Network 15: UNIT 01 PROCCESS
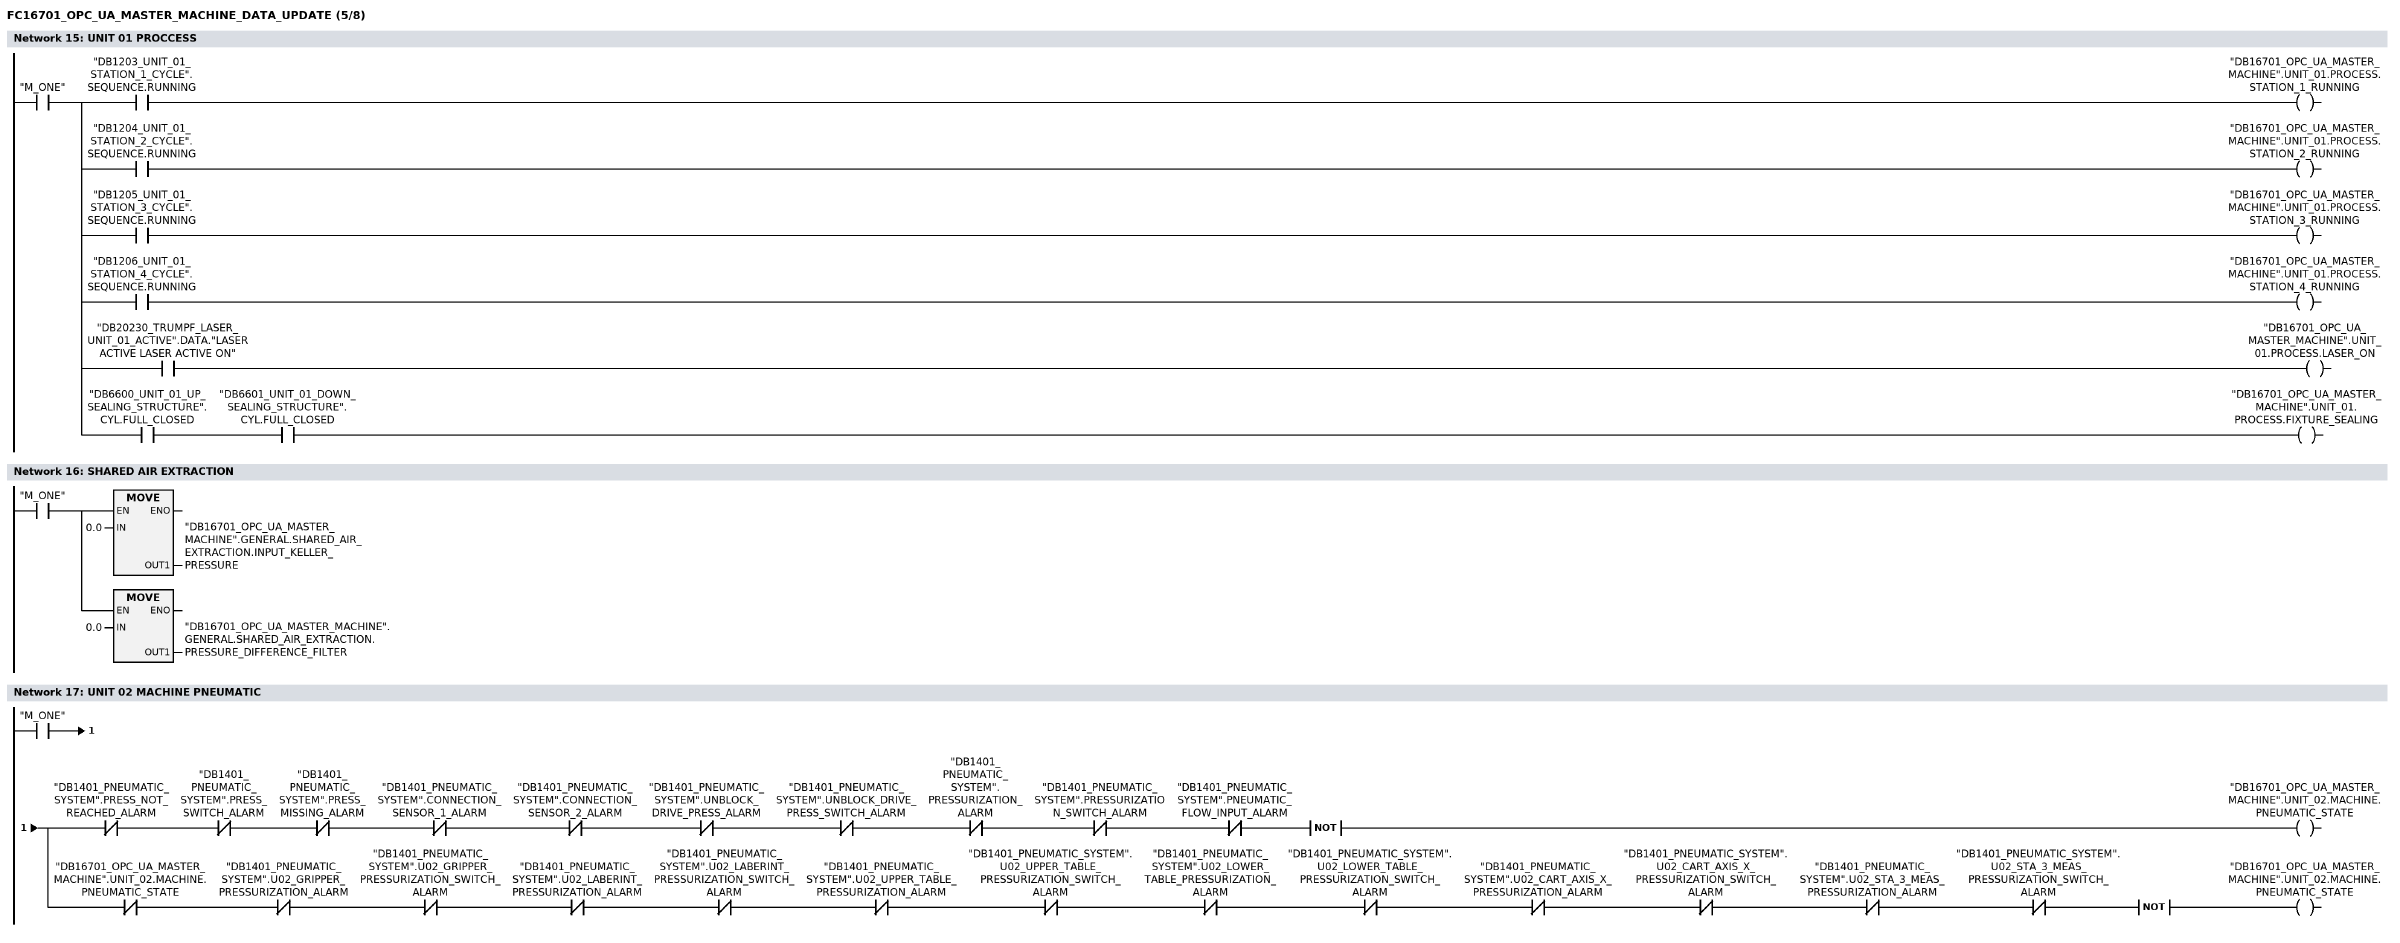
   RUNG wire#powerrail
      Contact( "M_ONE" )
      wire#w1
      Contact( "DB1203_UNIT_01_STATION_1_CYCLE".SEQUENCE.RUNNING )
      Coil( "DB16701_OPC_UA_MASTER_MACHINE".UNIT_01.PROCESS.STATION_1_RUNNING )
   END_RUNG
   RUNG wire#w1
      Contact( "DB1204_UNIT_01_STATION_2_CYCLE".SEQUENCE.RUNNING )
      Coil( "DB16701_OPC_UA_MASTER_MACHINE".UNIT_01.PROCESS.STATION_2_RUNNING )
   END_RUNG
   RUNG wire#w1
      Contact( "DB1205_UNIT_01_STATION_3_CYCLE".SEQUENCE.RUNNING )
      Coil( "DB16701_OPC_UA_MASTER_MACHINE".UNIT_01.PROCESS.STATION_3_RUNNING )
   END_RUNG
   RUNG wire#w1
      Contact( "DB1206_UNIT_01_STATION_4_CYCLE".SEQUENCE.RUNNING )
      Coil( "DB16701_OPC_UA_MASTER_MACHINE".UNIT_01.PROCESS.STATION_4_RUNNING )
   END_RUNG
   RUNG wire#w1
      Contact( "DB20230_TRUMPF_LASER_UNIT_01_ACTIVE".DATA."LASER ACTIVE LASER ACTIVE ON" )
      Coil( "DB16701_OPC_UA_MASTER_MACHINE".UNIT_01.PROCESS.LASER_ON )
   END_RUNG
   RUNG wire#w1
      Contact( "DB6600_UNIT_01_UP_SEALING_STRUCTURE".CYL.FULL_CLOSED )
      Contact( "DB6601_UNIT_01_DOWN_SEALING_STRUCTURE".CYL.FULL_CLOSED )
      Coil( "DB16701_OPC_UA_MASTER_MACHINE".UNIT_01.PROCESS.FIXTURE_SEALING )
   END_RUNG
   // the same network as SCL:
   "DB16701_OPC_UA_MASTER_MACHINE".UNIT_01.PROCESS.STATION_1_RUNNING := "M_ONE" AND "DB1203_UNIT_01_STATION_1_CYCLE".SEQUENCE.RUNNING;
   "DB16701_OPC_UA_MASTER_MACHINE".UNIT_01.PROCESS.STATION_2_RUNNING := "M_ONE" AND "DB1204_UNIT_01_STATION_2_CYCLE".SEQUENCE.RUNNING;
   "DB16701_OPC_UA_MASTER_MACHINE".UNIT_01.PROCESS.STATION_3_RUNNING := "M_ONE" AND "DB1205_UNIT_01_STATION_3_CYCLE".SEQUENCE.RUNNING;
   "DB16701_OPC_UA_MASTER_MACHINE".UNIT_01.PROCESS.STATION_4_RUNNING := "M_ONE" AND "DB1206_UNIT_01_STATION_4_CYCLE".SEQUENCE.RUNNING;
   "DB16701_OPC_UA_MASTER_MACHINE".UNIT_01.PROCESS.LASER_ON := "M_ONE" AND "DB20230_TRUMPF_LASER_UNIT_01_ACTIVE".DATA."LASER ACTIVE LASER ACTIVE ON";
   "DB16701_OPC_UA_MASTER_MACHINE".UNIT_01.PROCESS.FIXTURE_SEALING := "M_ONE" AND "DB6600_UNIT_01_UP_SEALING_STRUCTURE".CYL.FULL_CLOSED AND "DB6601_UNIT_01_DOWN_SEALING_STRUCTURE".CYL.FULL_CLOSED;
END_REGION

REGION Network 16: SHARED AIR EXTRACTION
   RUNG wire#powerrail
      Contact( "M_ONE" )
      wire#w1
      Move(in := 0.0, out1 => "DB16701_OPC_UA_MASTER_MACHINE".GENERAL.SHARED_AIR_EXTRACTION.INPUT_KELLER_PRESSURE)
   END_RUNG
   RUNG wire#w1
      Move(in := 0.0, out1 => "DB16701_OPC_UA_MASTER_MACHINE".GENERAL.SHARED_AIR_EXTRACTION.PRESSURE_DIFFERENCE_FILTER)
   END_RUNG
   // the same network as SCL:
   IF "M_ONE" THEN
       "DB16701_OPC_UA_MASTER_MACHINE".GENERAL.SHARED_AIR_EXTRACTION.INPUT_KELLER_PRESSURE := 0.0;
       "DB16701_OPC_UA_MASTER_MACHINE".GENERAL.SHARED_AIR_EXTRACTION.PRESSURE_DIFFERENCE_FILTER := 0.0;
   END_IF;
END_REGION

REGION Network 17: UNIT 02 MACHINE PNEUMATIC
   RUNG wire#powerrail
      Contact( "M_ONE" )
      wire#w1
      I_Contact( "DB1401_PNEUMATIC_SYSTEM".PRESS_NOT_REACHED_ALARM )
      I_Contact( "DB1401_PNEUMATIC_SYSTEM".PRESS_SWITCH_ALARM )
      I_Contact( "DB1401_PNEUMATIC_SYSTEM".PRESS_MISSING_ALARM )
      I_Contact( "DB1401_PNEUMATIC_SYSTEM".CONNECTION_SENSOR_1_ALARM )
      I_Contact( "DB1401_PNEUMATIC_SYSTEM".CONNECTION_SENSOR_2_ALARM )
      I_Contact( "DB1401_PNEUMATIC_SYSTEM".UNBLOCK_DRIVE_PRESS_ALARM )
      I_Contact( "DB1401_PNEUMATIC_SYSTEM".UNBLOCK_DRIVE_PRESS_SWITCH_ALARM )
      I_Contact( "DB1401_PNEUMATIC_SYSTEM".PRESSURIZATION_ALARM )
      I_Contact( "DB1401_PNEUMATIC_SYSTEM".PRESSURIZATION_SWITCH_ALARM )
      I_Contact( "DB1401_PNEUMATIC_SYSTEM".PNEUMATIC_FLOW_INPUT_ALARM )
      Not()
      Coil( "DB16701_OPC_UA_MASTER_MACHINE".UNIT_02.MACHINE.PNEUMATIC_STATE )
   END_RUNG
   RUNG wire#w1
      I_Contact( "DB16701_OPC_UA_MASTER_MACHINE".UNIT_02.MACHINE.PNEUMATIC_STATE )
      I_Contact( "DB1401_PNEUMATIC_SYSTEM".U02_GRIPPER_PRESSURIZATION_ALARM )
      I_Contact( "DB1401_PNEUMATIC_SYSTEM".U02_GRIPPER_PRESSURIZATION_SWITCH_ALARM )
      I_Contact( "DB1401_PNEUMATIC_SYSTEM".U02_LABERINT_PRESSURIZATION_ALARM )
      I_Contact( "DB1401_PNEUMATIC_SYSTEM".U02_LABERINT_PRESSURIZATION_SWITCH_ALARM )
      I_Contact( "DB1401_PNEUMATIC_SYSTEM".U02_UPPER_TABLE_PRESSURIZATION_ALARM )
      I_Contact( "DB1401_PNEUMATIC_SYSTEM".U02_UPPER_TABLE_PRESSURIZATION_SWITCH_ALARM )
      I_Contact( "DB1401_PNEUMATIC_SYSTEM".U02_LOWER_TABLE_PRESSURIZATION_ALARM )
      I_Contact( "DB1401_PNEUMATIC_SYSTEM".U02_LOWER_TABLE_PRESSURIZATION_SWITCH_ALARM )
      I_Contact( "DB1401_PNEUMATIC_SYSTEM".U02_CART_AXIS_X_PRESSURIZATION_ALARM )
      I_Contact( "DB1401_PNEUMATIC_SYSTEM".U02_CART_AXIS_X_PRESSURIZATION_SWITCH_ALARM )
      I_Contact( "DB1401_PNEUMATIC_SYSTEM".U02_STA_3_MEAS_PRESSURIZATION_ALARM )
      I_Contact( "DB1401_PNEUMATIC_SYSTEM".U02_STA_3_MEAS_PRESSURIZATION_SWITCH_ALARM )
      Not()
      Coil( "DB16701_OPC_UA_MASTER_MACHINE".UNIT_02.MACHINE.PNEUMATIC_STATE )
   END_RUNG
   // the same network as SCL:
   "DB16701_OPC_UA_MASTER_MACHINE".UNIT_02.MACHINE.PNEUMATIC_STATE := NOT ("M_ONE" AND NOT "DB1401_PNEUMATIC_SYSTEM".PRESS_NOT_REACHED_ALARM AND NOT "DB1401_PNEUMATIC_SYSTEM".PRESS_SWITCH_ALARM AND NOT "DB1401_PNEUMATIC_SYSTEM".PRESS_MISSING_ALARM AND NOT "DB1401_PNEUMATIC_SYSTEM".CONNECTION_SENSOR_1_ALARM AND NOT "DB1401_PNEUMATIC_SYSTEM".CONNECTION_SENSOR_2_ALARM AND NOT "DB1401_PNEUMATIC_SYSTEM".UNBLOCK_DRIVE_PRESS_ALARM AND NOT "DB1401_PNEUMATIC_SYSTEM".UNBLOCK_DRIVE_PRESS_SWITCH_ALARM AND NOT "DB1401_PNEUMATIC_SYSTEM".PRESSURIZATION_ALARM AND NOT "DB1401_PNEUMATIC_SYSTEM".PRESSURIZATION_SWITCH_ALARM AND NOT "DB1401_PNEUMATIC_SYSTEM".PNEUMATIC_FLOW_INPUT_ALARM);
   "DB16701_OPC_UA_MASTER_MACHINE".UNIT_02.MACHINE.PNEUMATIC_STATE := NOT ("M_ONE" AND NOT "DB16701_OPC_UA_MASTER_MACHINE".UNIT_02.MACHINE.PNEUMATIC_STATE AND NOT "DB1401_PNEUMATIC_SYSTEM".U02_GRIPPER_PRESSURIZATION_ALARM AND NOT "DB1401_PNEUMATIC_SYSTEM".U02_GRIPPER_PRESSURIZATION_SWITCH_ALARM AND NOT "DB1401_PNEUMATIC_SYSTEM".U02_LABERINT_PRESSURIZATION_ALARM AND NOT "DB1401_PNEUMATIC_SYSTEM".U02_LABERINT_PRESSURIZATION_SWITCH_ALARM AND NOT "DB1401_PNEUMATIC_SYSTEM".U02_UPPER_TABLE_PRESSURIZATION_ALARM AND NOT "DB1401_PNEUMATIC_SYSTEM".U02_UPPER_TABLE_PRESSURIZATION_SWITCH_ALARM AND NOT "DB1401_PNEUMATIC_SYSTEM".U02_LOWER_TABLE_PRESSURIZATION_ALARM AND NOT "DB1401_PNEUMATIC_SYSTEM".U02_LOWER_TABLE_PRESSURIZATION_SWITCH_ALARM AND NOT "DB1401_PNEUMATIC_SYSTEM".U02_CART_AXIS_X_PRESSURIZATION_ALARM AND NOT "DB1401_PNEUMATIC_SYSTEM".U02_CART_AXIS_X_PRESSURIZATION_SWITCH_ALARM AND NOT "DB1401_PNEUMATIC_SYSTEM".U02_STA_3_MEAS_PRESSURIZATION_ALARM AND NOT "DB1401_PNEUMATIC_SYSTEM".U02_STA_3_MEAS_PRESSURIZATION_SWITCH_ALARM);
END_REGION

REGION Network 18: UNIT 02 MACHINE TEMPERATURE
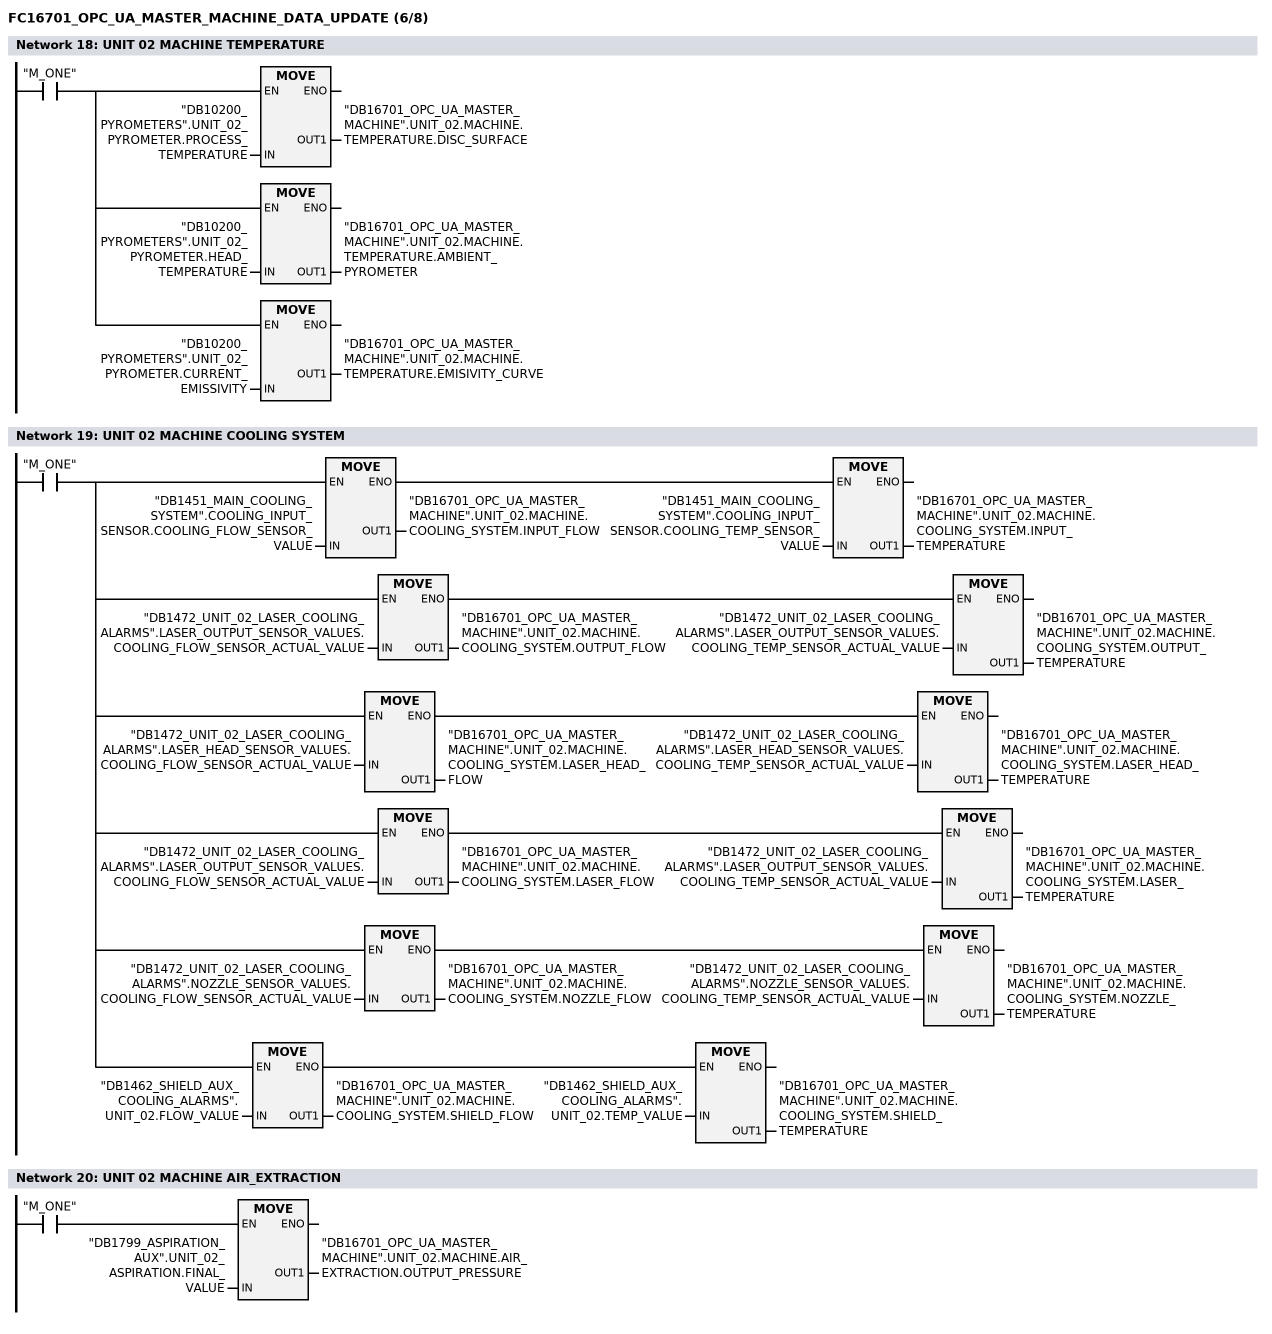
   RUNG wire#powerrail
      Contact( "M_ONE" )
      wire#w1
      Move(in := "DB10200_PYROMETERS".UNIT_02_PYROMETER.PROCESS_TEMPERATURE, out1 => "DB16701_OPC_UA_MASTER_MACHINE".UNIT_02.MACHINE.TEMPERATURE.DISC_SURFACE)
   END_RUNG
   RUNG wire#w1
      Move(in := "DB10200_PYROMETERS".UNIT_02_PYROMETER.HEAD_TEMPERATURE, out1 => "DB16701_OPC_UA_MASTER_MACHINE".UNIT_02.MACHINE.TEMPERATURE.AMBIENT_PYROMETER)
   END_RUNG
   RUNG wire#w1
      Move(in := "DB10200_PYROMETERS".UNIT_02_PYROMETER.CURRENT_EMISSIVITY, out1 => "DB16701_OPC_UA_MASTER_MACHINE".UNIT_02.MACHINE.TEMPERATURE.EMISIVITY_CURVE)
   END_RUNG
   // the same network as SCL:
   IF "M_ONE" THEN
       "DB16701_OPC_UA_MASTER_MACHINE".UNIT_02.MACHINE.TEMPERATURE.DISC_SURFACE := "DB10200_PYROMETERS".UNIT_02_PYROMETER.PROCESS_TEMPERATURE;
       "DB16701_OPC_UA_MASTER_MACHINE".UNIT_02.MACHINE.TEMPERATURE.AMBIENT_PYROMETER := "DB10200_PYROMETERS".UNIT_02_PYROMETER.HEAD_TEMPERATURE;
       "DB16701_OPC_UA_MASTER_MACHINE".UNIT_02.MACHINE.TEMPERATURE.EMISIVITY_CURVE := "DB10200_PYROMETERS".UNIT_02_PYROMETER.CURRENT_EMISSIVITY;
   END_IF;
END_REGION

REGION Network 19: UNIT 02 MACHINE COOLING SYSTEM
   RUNG wire#powerrail
      Contact( "M_ONE" )
      wire#w1
      Move(in := "DB1451_MAIN_COOLING_SYSTEM".COOLING_INPUT_SENSOR.COOLING_FLOW_SENSOR_VALUE, out1 => "DB16701_OPC_UA_MASTER_MACHINE".UNIT_02.MACHINE.COOLING_SYSTEM.INPUT_FLOW)
      Move(in := "DB1451_MAIN_COOLING_SYSTEM".COOLING_INPUT_SENSOR.COOLING_TEMP_SENSOR_VALUE, out1 => "DB16701_OPC_UA_MASTER_MACHINE".UNIT_02.MACHINE.COOLING_SYSTEM.INPUT_TEMPERATURE)
   END_RUNG
   RUNG wire#w1
      Move(in := "DB1472_UNIT_02_LASER_COOLING_ALARMS".LASER_OUTPUT_SENSOR_VALUES.COOLING_FLOW_SENSOR_ACTUAL_VALUE, out1 => "DB16701_OPC_UA_MASTER_MACHINE".UNIT_02.MACHINE.COOLING_SYSTEM.OUTPUT_FLOW)
      Move(in := "DB1472_UNIT_02_LASER_COOLING_ALARMS".LASER_OUTPUT_SENSOR_VALUES.COOLING_TEMP_SENSOR_ACTUAL_VALUE, out1 => "DB16701_OPC_UA_MASTER_MACHINE".UNIT_02.MACHINE.COOLING_SYSTEM.OUTPUT_TEMPERATURE)
   END_RUNG
   RUNG wire#w1
      Move(in := "DB1472_UNIT_02_LASER_COOLING_ALARMS".LASER_HEAD_SENSOR_VALUES.COOLING_FLOW_SENSOR_ACTUAL_VALUE, out1 => "DB16701_OPC_UA_MASTER_MACHINE".UNIT_02.MACHINE.COOLING_SYSTEM.LASER_HEAD_FLOW)
      Move(in := "DB1472_UNIT_02_LASER_COOLING_ALARMS".LASER_HEAD_SENSOR_VALUES.COOLING_TEMP_SENSOR_ACTUAL_VALUE, out1 => "DB16701_OPC_UA_MASTER_MACHINE".UNIT_02.MACHINE.COOLING_SYSTEM.LASER_HEAD_TEMPERATURE)
   END_RUNG
   RUNG wire#w1
      Move(in := "DB1472_UNIT_02_LASER_COOLING_ALARMS".LASER_OUTPUT_SENSOR_VALUES.COOLING_FLOW_SENSOR_ACTUAL_VALUE, out1 => "DB16701_OPC_UA_MASTER_MACHINE".UNIT_02.MACHINE.COOLING_SYSTEM.LASER_FLOW)
      Move(in := "DB1472_UNIT_02_LASER_COOLING_ALARMS".LASER_OUTPUT_SENSOR_VALUES.COOLING_TEMP_SENSOR_ACTUAL_VALUE, out1 => "DB16701_OPC_UA_MASTER_MACHINE".UNIT_02.MACHINE.COOLING_SYSTEM.LASER_TEMPERATURE)
   END_RUNG
   RUNG wire#w1
      Move(in := "DB1472_UNIT_02_LASER_COOLING_ALARMS".NOZZLE_SENSOR_VALUES.COOLING_FLOW_SENSOR_ACTUAL_VALUE, out1 => "DB16701_OPC_UA_MASTER_MACHINE".UNIT_02.MACHINE.COOLING_SYSTEM.NOZZLE_FLOW)
      Move(in := "DB1472_UNIT_02_LASER_COOLING_ALARMS".NOZZLE_SENSOR_VALUES.COOLING_TEMP_SENSOR_ACTUAL_VALUE, out1 => "DB16701_OPC_UA_MASTER_MACHINE".UNIT_02.MACHINE.COOLING_SYSTEM.NOZZLE_TEMPERATURE)
   END_RUNG
   RUNG wire#w1
      Move(in := "DB1462_SHIELD_AUX_COOLING_ALARMS".UNIT_02.FLOW_VALUE, out1 => "DB16701_OPC_UA_MASTER_MACHINE".UNIT_02.MACHINE.COOLING_SYSTEM.SHIELD_FLOW)
      Move(in := "DB1462_SHIELD_AUX_COOLING_ALARMS".UNIT_02.TEMP_VALUE, out1 => "DB16701_OPC_UA_MASTER_MACHINE".UNIT_02.MACHINE.COOLING_SYSTEM.SHIELD_TEMPERATURE)
   END_RUNG
   // the same network as SCL:
   IF "M_ONE" THEN
       "DB16701_OPC_UA_MASTER_MACHINE".UNIT_02.MACHINE.COOLING_SYSTEM.INPUT_FLOW := "DB1451_MAIN_COOLING_SYSTEM".COOLING_INPUT_SENSOR.COOLING_FLOW_SENSOR_VALUE;
       "DB16701_OPC_UA_MASTER_MACHINE".UNIT_02.MACHINE.COOLING_SYSTEM.INPUT_TEMPERATURE := "DB1451_MAIN_COOLING_SYSTEM".COOLING_INPUT_SENSOR.COOLING_TEMP_SENSOR_VALUE;
       "DB16701_OPC_UA_MASTER_MACHINE".UNIT_02.MACHINE.COOLING_SYSTEM.OUTPUT_FLOW := "DB1472_UNIT_02_LASER_COOLING_ALARMS".LASER_OUTPUT_SENSOR_VALUES.COOLING_FLOW_SENSOR_ACTUAL_VALUE;
       "DB16701_OPC_UA_MASTER_MACHINE".UNIT_02.MACHINE.COOLING_SYSTEM.OUTPUT_TEMPERATURE := "DB1472_UNIT_02_LASER_COOLING_ALARMS".LASER_OUTPUT_SENSOR_VALUES.COOLING_TEMP_SENSOR_ACTUAL_VALUE;
       "DB16701_OPC_UA_MASTER_MACHINE".UNIT_02.MACHINE.COOLING_SYSTEM.LASER_HEAD_FLOW := "DB1472_UNIT_02_LASER_COOLING_ALARMS".LASER_HEAD_SENSOR_VALUES.COOLING_FLOW_SENSOR_ACTUAL_VALUE;
       "DB16701_OPC_UA_MASTER_MACHINE".UNIT_02.MACHINE.COOLING_SYSTEM.LASER_HEAD_TEMPERATURE := "DB1472_UNIT_02_LASER_COOLING_ALARMS".LASER_HEAD_SENSOR_VALUES.COOLING_TEMP_SENSOR_ACTUAL_VALUE;
       "DB16701_OPC_UA_MASTER_MACHINE".UNIT_02.MACHINE.COOLING_SYSTEM.LASER_FLOW := "DB1472_UNIT_02_LASER_COOLING_ALARMS".LASER_OUTPUT_SENSOR_VALUES.COOLING_FLOW_SENSOR_ACTUAL_VALUE;
       "DB16701_OPC_UA_MASTER_MACHINE".UNIT_02.MACHINE.COOLING_SYSTEM.LASER_TEMPERATURE := "DB1472_UNIT_02_LASER_COOLING_ALARMS".LASER_OUTPUT_SENSOR_VALUES.COOLING_TEMP_SENSOR_ACTUAL_VALUE;
       "DB16701_OPC_UA_MASTER_MACHINE".UNIT_02.MACHINE.COOLING_SYSTEM.NOZZLE_FLOW := "DB1472_UNIT_02_LASER_COOLING_ALARMS".NOZZLE_SENSOR_VALUES.COOLING_FLOW_SENSOR_ACTUAL_VALUE;
       "DB16701_OPC_UA_MASTER_MACHINE".UNIT_02.MACHINE.COOLING_SYSTEM.NOZZLE_TEMPERATURE := "DB1472_UNIT_02_LASER_COOLING_ALARMS".NOZZLE_SENSOR_VALUES.COOLING_TEMP_SENSOR_ACTUAL_VALUE;
       "DB16701_OPC_UA_MASTER_MACHINE".UNIT_02.MACHINE.COOLING_SYSTEM.SHIELD_FLOW := "DB1462_SHIELD_AUX_COOLING_ALARMS".UNIT_02.FLOW_VALUE;
       "DB16701_OPC_UA_MASTER_MACHINE".UNIT_02.MACHINE.COOLING_SYSTEM.SHIELD_TEMPERATURE := "DB1462_SHIELD_AUX_COOLING_ALARMS".UNIT_02.TEMP_VALUE;
   END_IF;
END_REGION

REGION Network 20: UNIT 02 MACHINE AIR_EXTRACTION
   RUNG wire#powerrail
      Contact( "M_ONE" )
      Move(in := "DB1799_ASPIRATION_AUX".UNIT_02_ASPIRATION.FINAL_VALUE, out1 => "DB16701_OPC_UA_MASTER_MACHINE".UNIT_02.MACHINE.AIR_EXTRACTION.OUTPUT_PRESSURE)
   END_RUNG
   // the same network as SCL:
   IF "M_ONE" THEN
       "DB16701_OPC_UA_MASTER_MACHINE".UNIT_02.MACHINE.AIR_EXTRACTION.OUTPUT_PRESSURE := "DB1799_ASPIRATION_AUX".UNIT_02_ASPIRATION.FINAL_VALUE;
   END_IF;
END_REGION

REGION Network 21: UNIT 02 MACHINE ST3 PRESSURE CONTROL
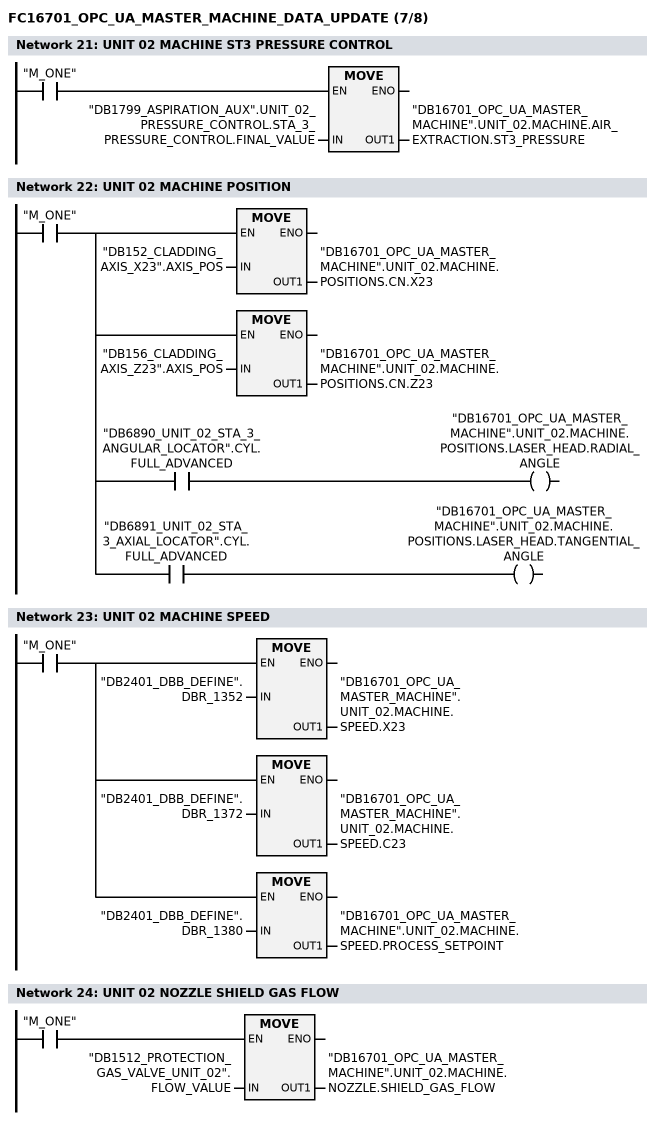
   RUNG wire#powerrail
      Contact( "M_ONE" )
      Move(in := "DB1799_ASPIRATION_AUX".UNIT_02_PRESSURE_CONTROL.STA_3_PRESSURE_CONTROL.FINAL_VALUE, out1 => "DB16701_OPC_UA_MASTER_MACHINE".UNIT_02.MACHINE.AIR_EXTRACTION.ST3_PRESSURE)
   END_RUNG
   // the same network as SCL:
   IF "M_ONE" THEN
       "DB16701_OPC_UA_MASTER_MACHINE".UNIT_02.MACHINE.AIR_EXTRACTION.ST3_PRESSURE := "DB1799_ASPIRATION_AUX".UNIT_02_PRESSURE_CONTROL.STA_3_PRESSURE_CONTROL.FINAL_VALUE;
   END_IF;
END_REGION

REGION Network 22: UNIT 02 MACHINE POSITION
   RUNG wire#powerrail
      Contact( "M_ONE" )
      wire#w1
      Move(in := "DB152_CLADDING_AXIS_X23".AXIS_POS, out1 => "DB16701_OPC_UA_MASTER_MACHINE".UNIT_02.MACHINE.POSITIONS.CN.X23)
   END_RUNG
   RUNG wire#w1
      Move(in := "DB156_CLADDING_AXIS_Z23".AXIS_POS, out1 => "DB16701_OPC_UA_MASTER_MACHINE".UNIT_02.MACHINE.POSITIONS.CN.Z23)
   END_RUNG
   RUNG wire#w1
      Contact( "DB6890_UNIT_02_STA_3_ANGULAR_LOCATOR".CYL.FULL_ADVANCED )
      Coil( "DB16701_OPC_UA_MASTER_MACHINE".UNIT_02.MACHINE.POSITIONS.LASER_HEAD.RADIAL_ANGLE )
   END_RUNG
   RUNG wire#w1
      Contact( "DB6891_UNIT_02_STA_3_AXIAL_LOCATOR".CYL.FULL_ADVANCED )
      Coil( "DB16701_OPC_UA_MASTER_MACHINE".UNIT_02.MACHINE.POSITIONS.LASER_HEAD.TANGENTIAL_ANGLE )
   END_RUNG
   // the same network as SCL:
   IF "M_ONE" THEN
       "DB16701_OPC_UA_MASTER_MACHINE".UNIT_02.MACHINE.POSITIONS.CN.X23 := "DB152_CLADDING_AXIS_X23".AXIS_POS;
       "DB16701_OPC_UA_MASTER_MACHINE".UNIT_02.MACHINE.POSITIONS.CN.Z23 := "DB156_CLADDING_AXIS_Z23".AXIS_POS;
   END_IF;
   "DB16701_OPC_UA_MASTER_MACHINE".UNIT_02.MACHINE.POSITIONS.LASER_HEAD.RADIAL_ANGLE := "M_ONE" AND "DB6890_UNIT_02_STA_3_ANGULAR_LOCATOR".CYL.FULL_ADVANCED;
   "DB16701_OPC_UA_MASTER_MACHINE".UNIT_02.MACHINE.POSITIONS.LASER_HEAD.TANGENTIAL_ANGLE := "M_ONE" AND "DB6891_UNIT_02_STA_3_AXIAL_LOCATOR".CYL.FULL_ADVANCED;
END_REGION

REGION Network 23: UNIT 02 MACHINE SPEED
   RUNG wire#powerrail
      Contact( "M_ONE" )
      wire#w1
      Move(in := "DB2401_DBB_DEFINE".DBR_1352, out1 => "DB16701_OPC_UA_MASTER_MACHINE".UNIT_02.MACHINE.SPEED.X23)
   END_RUNG
   RUNG wire#w1
      Move(in := "DB2401_DBB_DEFINE".DBR_1372, out1 => "DB16701_OPC_UA_MASTER_MACHINE".UNIT_02.MACHINE.SPEED.C23)
   END_RUNG
   RUNG wire#w1
      Move(in := "DB2401_DBB_DEFINE".DBR_1380, out1 => "DB16701_OPC_UA_MASTER_MACHINE".UNIT_02.MACHINE.SPEED.PROCESS_SETPOINT)
   END_RUNG
   // the same network as SCL:
   IF "M_ONE" THEN
       "DB16701_OPC_UA_MASTER_MACHINE".UNIT_02.MACHINE.SPEED.X23 := "DB2401_DBB_DEFINE".DBR_1352;
       "DB16701_OPC_UA_MASTER_MACHINE".UNIT_02.MACHINE.SPEED.C23 := "DB2401_DBB_DEFINE".DBR_1372;
       "DB16701_OPC_UA_MASTER_MACHINE".UNIT_02.MACHINE.SPEED.PROCESS_SETPOINT := "DB2401_DBB_DEFINE".DBR_1380;
   END_IF;
END_REGION

REGION Network 24: UNIT 02 NOZZLE SHIELD GAS FLOW
   RUNG wire#powerrail
      Contact( "M_ONE" )
      Move(in := "DB1512_PROTECTION_GAS_VALVE_UNIT_02".FLOW_VALUE, out1 => "DB16701_OPC_UA_MASTER_MACHINE".UNIT_02.MACHINE.NOZZLE.SHIELD_GAS_FLOW)
   END_RUNG
   // the same network as SCL:
   IF "M_ONE" THEN
       "DB16701_OPC_UA_MASTER_MACHINE".UNIT_02.MACHINE.NOZZLE.SHIELD_GAS_FLOW := "DB1512_PROTECTION_GAS_VALVE_UNIT_02".FLOW_VALUE;
   END_IF;
END_REGION

REGION Network 25: UNIT 02 PROCCESS
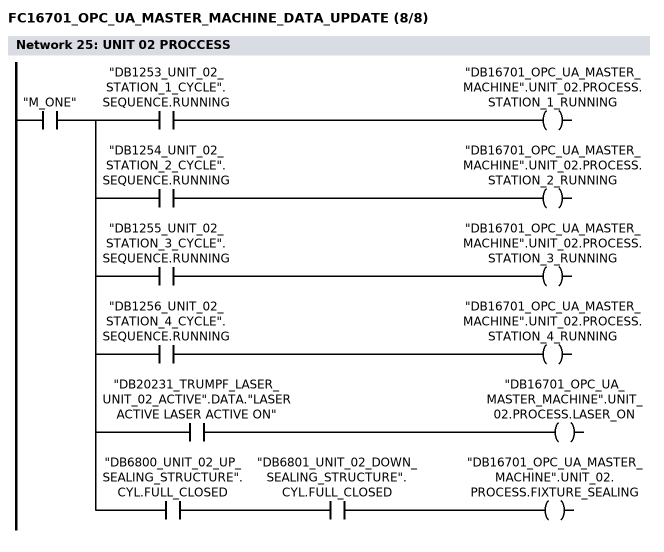
   RUNG wire#powerrail
      Contact( "M_ONE" )
      wire#w1
      Contact( "DB1253_UNIT_02_STATION_1_CYCLE".SEQUENCE.RUNNING )
      Coil( "DB16701_OPC_UA_MASTER_MACHINE".UNIT_02.PROCESS.STATION_1_RUNNING )
   END_RUNG
   RUNG wire#w1
      Contact( "DB1254_UNIT_02_STATION_2_CYCLE".SEQUENCE.RUNNING )
      Coil( "DB16701_OPC_UA_MASTER_MACHINE".UNIT_02.PROCESS.STATION_2_RUNNING )
   END_RUNG
   RUNG wire#w1
      Contact( "DB1255_UNIT_02_STATION_3_CYCLE".SEQUENCE.RUNNING )
      Coil( "DB16701_OPC_UA_MASTER_MACHINE".UNIT_02.PROCESS.STATION_3_RUNNING )
   END_RUNG
   RUNG wire#w1
      Contact( "DB1256_UNIT_02_STATION_4_CYCLE".SEQUENCE.RUNNING )
      Coil( "DB16701_OPC_UA_MASTER_MACHINE".UNIT_02.PROCESS.STATION_4_RUNNING )
   END_RUNG
   RUNG wire#w1
      Contact( "DB20231_TRUMPF_LASER_UNIT_02_ACTIVE".DATA."LASER ACTIVE LASER ACTIVE ON" )
      Coil( "DB16701_OPC_UA_MASTER_MACHINE".UNIT_02.PROCESS.LASER_ON )
   END_RUNG
   RUNG wire#w1
      Contact( "DB6800_UNIT_02_UP_SEALING_STRUCTURE".CYL.FULL_CLOSED )
      Contact( "DB6801_UNIT_02_DOWN_SEALING_STRUCTURE".CYL.FULL_CLOSED )
      Coil( "DB16701_OPC_UA_MASTER_MACHINE".UNIT_02.PROCESS.FIXTURE_SEALING )
   END_RUNG
   // the same network as SCL:
   "DB16701_OPC_UA_MASTER_MACHINE".UNIT_02.PROCESS.STATION_1_RUNNING := "M_ONE" AND "DB1253_UNIT_02_STATION_1_CYCLE".SEQUENCE.RUNNING;
   "DB16701_OPC_UA_MASTER_MACHINE".UNIT_02.PROCESS.STATION_2_RUNNING := "M_ONE" AND "DB1254_UNIT_02_STATION_2_CYCLE".SEQUENCE.RUNNING;
   "DB16701_OPC_UA_MASTER_MACHINE".UNIT_02.PROCESS.STATION_3_RUNNING := "M_ONE" AND "DB1255_UNIT_02_STATION_3_CYCLE".SEQUENCE.RUNNING;
   "DB16701_OPC_UA_MASTER_MACHINE".UNIT_02.PROCESS.STATION_4_RUNNING := "M_ONE" AND "DB1256_UNIT_02_STATION_4_CYCLE".SEQUENCE.RUNNING;
   "DB16701_OPC_UA_MASTER_MACHINE".UNIT_02.PROCESS.LASER_ON := "M_ONE" AND "DB20231_TRUMPF_LASER_UNIT_02_ACTIVE".DATA."LASER ACTIVE LASER ACTIVE ON";
   "DB16701_OPC_UA_MASTER_MACHINE".UNIT_02.PROCESS.FIXTURE_SEALING := "M_ONE" AND "DB6800_UNIT_02_UP_SEALING_STRUCTURE".CYL.FULL_CLOSED AND "DB6801_UNIT_02_DOWN_SEALING_STRUCTURE".CYL.FULL_CLOSED;
END_REGION
END_FUNCTION
